// TwinCAT 3 PLC project TcAocLib
// Title: CNM AoC Lib
// Company: ekvip automation GmbH
// Author: tdie
// ProjectVersion: 0.0.0.0
// ProgramVersion: 3.1.4026.11
// libraries:
//   CNM_AbstractObject, * (ekvip automation GmbH)
//   CNM_AssertionInterfaceLib, * (ekvip automation GmbH)
//   CNM_CollectionInterfaces, * (ekvip automation GmbH)
//   CNM_Collections, * (ekvip automation GmbH)
//   CNM_CycleManager, * (ekvip automation GmbH)
//   CNM_CylceManagerInterfaces, * (ekvip automation GmbH)
//   CNM_ReturnTypes, * (ekvip automation GmbH)
//   CNM_UnicodeUtilities, * (ekvip automation GmbH)
//   Tc2_Standard, * (Beckhoff Automation GmbH)
//   Tc2_System, * (Beckhoff Automation GmbH)
//   Tc2_Utilities, * (Beckhoff Automation GmbH)
// project tree:
//   File/ FileHandler.TcPOU
//   Project Information/ F_GetCompany.TcPOU, F_GetTitle.TcPOU, F_GetVersion.TcPOU
//   Solver/ AbstractSolver.TcPOU
//   Strings/ GetAllLinesFromString.TcPOU, ILine.TcIO, IStringContainer.TcIO, Line.TcPOU
//   Strings/Wrapper/ ILineList.TcIO, IStringContainerList.TcIO, LineList.TcPOU, StringContainerList.TcPOU
//   Value/ IHaveUlintValue.TcIO, IHaveValue.TcIO, IHaveLintValue.TcIO, UlintValue.TcPOU, Value.TcPOU, ValueSum.TcPOU, LintValue.TcPOU
//   Version/ Global_Version.TcGVL
// (motion and I/O tree: see PLC project solutions)
// real-time tasks:
//   TASK PlcTask: cycle T#10ms, priority 20, ADS port 350

// ---- Version/Global_Version.TcGVL
{attribute 'TcGenerated'}
{attribute 'no-analysis'}
{attribute 'linkalways'}
// This function has been automatically generated from the project information.
VAR_GLOBAL CONSTANT
	{attribute 'const_non_replaced'}
	stLibVersion_CNM_AoC_Lib : ST_LibVersion := (iMajor := 0, iMinor := 0, iBuild := 0, iRevision := 0, nFlags := 0, sVersion := '0.0.0.0');
END_VAR

// ---- Strings/ILine.TcIO
INTERFACE ILine EXTENDS IStringContainer

METHOD splitBy : IStringContainerList
VAR_INPUT
	splitter	: STRING(255);
	addEmptyEntries :BOOL := FALSE;
END_VAR
END_METHOD

END_INTERFACE

// ---- Strings/IStringContainer.TcIO
INTERFACE IStringContainer EXTENDS IHaveValue

PROPERTY text : STRING(255)
GET
END_GET
SET
END_SET
END_PROPERTY

END_INTERFACE

// ---- Strings/Wrapper/ILineList.TcIO
INTERFACE ILineList EXTENDS CNM_AbstractObject.IObject

(*

short summary
=================
This methode adds the given CNM_AbstractObject.IObject to the end of the list.
Example: 
Given a list that looks like this: (Head->) A B C (<- End),
calling append(D) on this list will place the D at the and,
making it the new End: (Head->) A B C D(<- End)

.. <legal notes>

legal notes
=================
| SPDX-FileCopyrightText: © 2022 ekvip automation GmbH <info@ekvip.de>
| SPDX-License-Identifier: Apache-2.0
| For details check: Apache-2.0_

.. _Apache-2.0: https://www.apache.org/licenses/LICENSE-2.0

.. </legal notes>

parameters
=================

*)
METHOD append : CNM_CollectionInterfaces.CNM_ReturnTypes.SingleExecutionResult
VAR_INPUT
	(*The object to be appended*)
	line	: ILine;
END_VAR
END_METHOD

{warning 'Add method implementation '}
(*

short summary
=================
This methode adds all elements of the given collection to the end of this list.
Example:
For the list1: A B C and list2: D E F will be after list1.appendCollection(list2):
A B C D E F. Notice the elements are still in the same order they where befor on each subsection.

.. <legal notes>

legal notes
=================
| SPDX-FileCopyrightText: © 2022 ekvip automation GmbH <info@ekvip.de>
| SPDX-License-Identifier: Apache-2.0
| For details check: Apache-2.0_

.. _Apache-2.0: https://www.apache.org/licenses/LICENSE-2.0

.. </legal notes>

parameters
=================

*)
METHOD appendCollection : CNM_CollectionInterfaces.CNM_ReturnTypes.SingleExecutionResult
VAR_INPUT
	(*The collection to be appended*)
	collectionToAppend	: CNM_CollectionInterfaces.ICollection;
END_VAR
END_METHOD

{warning 'Add method implementation '}
(*

short summary
=================
This methode clears/deletes all clearable data from this object.
Example:
A list: 1 2 3 after list.clear() will have no remaining items, isEmpty = true.

.. <legal notes>

legal notes
=================
| SPDX-FileCopyrightText: © 2022 ekvip automation GmbH <info@ekvip.de>
| SPDX-License-Identifier: Apache-2.0
| For details check: Apache-2.0_

.. _Apache-2.0: https://www.apache.org/licenses/LICENSE-2.0

.. </legal notes>

parameters
=================

*)
METHOD clear
END_METHOD

{warning 'Add method implementation '}
(*

short summary
=================
This methode checks if a given object is contained in the collection. 
The object is inside if the collection contains an object where the default comperator of the objects returns EQUAL on compareTo!

.. <legal notes>

legal notes
=================
| SPDX-FileCopyrightText: © 2022 ekvip automation GmbH <info@ekvip.de>
| SPDX-License-Identifier: Apache-2.0
| For details check: Apache-2.0_

.. _Apache-2.0: https://www.apache.org/licenses/LICENSE-2.0

.. </legal notes>

parameters
=================
:return: ``FALSE``: list does not contain an equal object
    ``TRUE``: list does contain an equal object

*)
METHOD containsEqualLine : BOOL
VAR_INPUT
	(*the object to be checked if it exists inside the collection*)
	line	: ILine;
END_VAR
END_METHOD

{warning 'Add method implementation '}
(*

short summary
=================
This methode checks if a given object is contained in the collection. 
The object is inside if the collection contains an object of equal hashcode!

.. <legal notes>

legal notes
=================
| SPDX-FileCopyrightText: © 2022 ekvip automation GmbH <info@ekvip.de>
| SPDX-License-Identifier: Apache-2.0
| For details check: Apache-2.0_

.. _Apache-2.0: https://www.apache.org/licenses/LICENSE-2.0

.. </legal notes>

parameters
=================
:return: ``FALSE``: list does not contain given object,
    ``TRUE``: list does contain given object

*)
METHOD containsLine : BOOL
VAR_INPUT
	(*the object to be checked if it exists inside the collection*)
	line	: ILine;
END_VAR
END_METHOD

{warning 'Add method implementation '}
(*

short summary
=================
This property returns the last object in the first and removes it from the list. Can be seen as opposite of prepend.
Example:
On a list: (Head -->) A B C, list.dequeue will return A.
Example 2:
If you call prepend(x), a dequeue right after will return x.

.. <legal notes>

legal notes
=================
| SPDX-FileCopyrightText: © 2022 ekvip automation GmbH <info@ekvip.de>
| SPDX-License-Identifier: Apache-2.0
| For details check: Apache-2.0_

.. _Apache-2.0: https://www.apache.org/licenses/LICENSE-2.0

.. </legal notes>

*)
METHOD dequeue : ILine
END_METHOD

{warning 'Add method implementation '}
(*

short summary
=================
Method to perform a given action on all objects inside the collection.
Needs to reset the execution flag between calls.
Action to perform needs to implement :ref:`IApplier`.
Example:
You have a list of numbers: 1 2 3 and a ConcreteIncrementApplier that can take  a number and increment it. 
Calling list.forEach(TRUE, ConcreteIncrementApplier) will increment all numbers in the list, becoming: 2 3 4.

.. <legal notes>

legal notes
=================
| SPDX-FileCopyrightText: © 2022 ekvip automation GmbH <info@ekvip.de>
| SPDX-License-Identifier: Apache-2.0
| For details check: Apache-2.0_

.. _Apache-2.0: https://www.apache.org/licenses/LICENSE-2.0

.. </legal notes>

parameters
=========================
:return: CNM_ReturnTypes.ExecutionState

*)
METHOD forEach : CNM_CollectionInterfaces.CNM_ReturnTypes.SingleExecutionState
VAR_INPUT
	(*control bit to start or abort the forEach loop*)
	execute	: BOOL;
	(*the applier (action) to be used on all obejcts in the collection*)
	applier	: CNM_CollectionInterfaces.IApplier;
END_VAR
END_METHOD

{warning 'Add method implementation '}
(*

short summary
=================
This methode returns ths index of the first object that is equal to the given.
Example:
A list of: 1 2 3 after list.getIndexOf(1) will return: index=>0 and return IndexBounds.IN_BOUNDS
Example 2:
A list of: 1 2 3 after list.getIndexOf(4) will return: index=>3 and return IndexBounds.OUT_OF_BOUNDS

.. <legal notes>

legal notes
=================
| SPDX-FileCopyrightText: © 2022 ekvip automation GmbH <info@ekvip.de>
| SPDX-License-Identifier: Apache-2.0
| For details check: Apache-2.0_

.. _Apache-2.0: https://www.apache.org/licenses/LICENSE-2.0

.. </legal notes>

parameters
=================
:return: ``SingleExecutionResult.SUCCESS``: object found
    ``SingleExecutionResult.ERROR``: object couldn't be found in the list, index is undefined

*)
METHOD getIndexOf : CNM_CollectionInterfaces.CNM_ReturnTypes.SingleExecutionResult
VAR_INPUT
	(*the object to get the index from*)
	line	: ILine;
END_VAR
VAR_OUTPUT
	(*the index of the object inside the collection*)
	index	: __XWORD;
END_VAR
END_METHOD

{warning 'Add method implementation '}
(*

short summary
=================
This methode returns the object at the given index.
Returned objects can be modified, but not replaced! To replace an object use replaceObjectAt.
Example:
A list of: 1 2 3 after list.getObjectAt(1) will return: object=>2 and return SingleExecutionResult.SUCCESS
Example 2:
A list of: 1 2 3 after list.getObjectAt(3) will return: object=>NULL and return SingleExecutionResult.ERROR

.. <legal notes>

legal notes
=================
| SPDX-FileCopyrightText: © 2022 ekvip automation GmbH <info@ekvip.de>
| SPDX-License-Identifier: Apache-2.0
| For details check: Apache-2.0_

.. _Apache-2.0: https://www.apache.org/licenses/LICENSE-2.0

.. </legal notes>

parameters
=================
:return: ``SingleExecutionResult.SUCCESS``: index was valid
    ``SingleExecutionResult.ERROR``: index was not valid, returned object is undefined

*)
METHOD getLineAt : CNM_CollectionInterfaces.CNM_ReturnTypes.SingleExecutionResult
VAR_INPUT
	(*the index to access the object from*)
	index	: __XWORD;
END_VAR
VAR_OUTPUT
	(*the object at the given index*)
	line	: ILine;
END_VAR
END_METHOD

{warning 'Add property implementation'}
(*

short summary
=================
This property returns ``TRUE`` if the collection has any element.

.. <legal notes>

legal notes
=================
| SPDX-FileCopyrightText: © 2022 ekvip automation GmbH <info@ekvip.de>
| SPDX-License-Identifier: Apache-2.0
| For details check: Apache-2.0_

.. _Apache-2.0: https://www.apache.org/licenses/LICENSE-2.0

.. </legal notes>

*)
PROPERTY hasElement : BOOL
GET
END_GET
END_PROPERTY

{warning 'Add method implementation '}
(*

short summary
=================
This methode adds the given object at the given index. 
Will shift the other data starting at given index to the right.
List Lenght will be incremented.
Example:
A list of: 1 2 3 after list.insertObjectAt(1, object:=4) will become: 1 4 2 3 and return SingleExecutionResult.SUCCESS
Example 2:
A list of: 1 2 3 after list.insertObjectAt(3, object:=4) will become: 1 2 3 4 and return SingleExecutionResult.SUCCESS
Example 3:
A list of: 1 2 3 after list.insertObjectAt(5, object:=4) will become: 1 2 3 and return SingleExecutionResult.ERROR

.. <legal notes>

legal notes
=================
| SPDX-FileCopyrightText: © 2022 ekvip automation GmbH <info@ekvip.de>
| SPDX-License-Identifier: Apache-2.0
| For details check: Apache-2.0_

.. _Apache-2.0: https://www.apache.org/licenses/LICENSE-2.0

.. </legal notes>

parameters
=================
:return: ``SingleExecutionResult.SUCCESS``: index was valid, object inserted
    ``SingleExecutionResult.ERROR``: index out of bounds, list not changed

*)
METHOD insertLineAt : CNM_CollectionInterfaces.CNM_ReturnTypes.SingleExecutionResult
VAR_INPUT
	(*the index to insert the object at*)
	index	: __XWORD;
	(*the object to be added*)
	line	: ILine;
END_VAR
END_METHOD

{warning 'Add method implementation '}
(*

short summary
=================
This method sorts the Sortable in the inverted order, so from great to low
.. <legal notes>

legal notes
=================
| SPDX-FileCopyrightText: © 2022 ekvip automation GmbH <info@ekvip.de>
| SPDX-License-Identifier: Apache-2.0
| For details check: Apache-2.0_

.. _Apache-2.0: https://www.apache.org/licenses/LICENSE-2.0

.. </legal notes>

parameters
=========================
:return: ``ABORTED``: While inverse was pending,execute had a falling edge,
	``BUSY``: Inverse is in progress
	``ERROR``: Inverse was not able to finish (p.e. List changed) call inverse(false) to reset
	``IDLE``: Currently invert is not in progress
	``SUCCESS``: Inversing was finished 
*)
METHOD inverseSort : CNM_CollectionInterfaces.CNM_ReturnTypes.SingleExecutionState
VAR_INPUT
	(*control bit to start or abort the inverting, needs to be active until the ExecutionState is noz longer busy*)
	execute	: BOOL;
END_VAR
END_METHOD

{warning 'Add method implementation '}
(*

short summary
=================
Inverts the order of the elements inside the object. Does not apply any kind of sorting, only reverses.

.. <legal notes>

legal notes
=================
| SPDX-FileCopyrightText: © 2022 ekvip automation GmbH <info@ekvip.de>
| SPDX-License-Identifier: Apache-2.0
| For details check: Apache-2.0_

.. _Apache-2.0: https://www.apache.org/licenses/LICENSE-2.0

.. </legal notes>

parameters
=========================

*)
METHOD invert
END_METHOD

{warning 'Add property implementation'}
(*

short summary
=================
This property returns ``TRUE`` if the collection is empty.

.. <legal notes>

legal notes
=================
| SPDX-FileCopyrightText: © 2022 ekvip automation GmbH <info@ekvip.de>
| SPDX-License-Identifier: Apache-2.0
| For details check: Apache-2.0_

.. _Apache-2.0: https://www.apache.org/licenses/LICENSE-2.0

.. </legal notes>

*)
PROPERTY isEmpty : BOOL
GET
END_GET
END_PROPERTY

{warning 'Add method implementation '}
(*

short summary
=================
This methode returns the next object in the iteration and returns an execution state.
Example:
You have a list: 1 2 3
the first iterate call will return CNM_ReturnTypes.BUSY and object = 1
the second iterate call will return CNM_ReturnTypes.BUSY and object = 2
the third iterate call will return CNM_ReturnTypes.SUCCESS and object = 3

.. <legal notes>

legal notes
=================
| SPDX-FileCopyrightText: © 2022 ekvip automation GmbH <info@ekvip.de>
| SPDX-License-Identifier: Apache-2.0
| For details check: Apache-2.0_

.. _Apache-2.0: https://www.apache.org/licenses/LICENSE-2.0

.. </legal notes>

parameters
=================

*)
METHOD iterate : CNM_CollectionInterfaces.CNM_ReturnTypes.SingleExecutionState
VAR_INPUT
	(*control bit to start or abort the iterate*)
	execute	: BOOL;
END_VAR
VAR_OUTPUT
	(*the returned object of the iteration*)
	line	: ILine;
END_VAR
END_METHOD

{warning 'Add method implementation '}
(*

short summary
=================
This property returns the last object in the list and removes it from the list. Can be seen as opposite of append.
Example:
On a list: (Head -->) A B C, list.pop will return C.
Example 2:
If you call append(x), a pop right after will return x.
May return a null pointer if list is empty

.. <legal notes>

legal notes
=================
| SPDX-FileCopyrightText: © 2022 ekvip automation GmbH <info@ekvip.de>
| SPDX-License-Identifier: Apache-2.0
| For details check: Apache-2.0_

.. _Apache-2.0: https://www.apache.org/licenses/LICENSE-2.0

.. </legal notes>

*)
METHOD pop : ILine
END_METHOD

{warning 'Add method implementation '}
(*

short summary
=================
This methode adds the given obejct to the end of the list.
Example: 
Given a list that looks like this: (Head->) A B C (<- End),
calling prepend(D) on this list will place the D at start,
making it the new Head: (Head->) D A B C (<- End)

.. <legal notes>

legal notes
=================
| SPDX-FileCopyrightText: © 2022 ekvip automation GmbH <info@ekvip.de>
| SPDX-License-Identifier: Apache-2.0
| For details check: Apache-2.0_

.. _Apache-2.0: https://www.apache.org/licenses/LICENSE-2.0

.. </legal notes>

parameters
=================
:return: ``SingleExecutionResult.SUCCESS``: prepend was successful
	``SingleExecutionResult.ERROR``: allocation of memory for new object failed
	
*)
METHOD prepend : CNM_CollectionInterfaces.CNM_ReturnTypes.SingleExecutionResult
VAR_INPUT
	(*The object to be prepended*)
	line	: ILine;
END_VAR
END_METHOD

{warning 'Add method implementation '}
(*

short summary
=================
This methode adds all elements of the given collection to the start of this list. 
Example:
For the list1: A B C and list2: D E F will be after list1.prependCollection(list2):
D E F A B C. Notice the elements are still in the same order they where befor on each subsection.

.. <legal notes>

legal notes
=================
| SPDX-FileCopyrightText: © 2022 ekvip automation GmbH <info@ekvip.de>
| SPDX-License-Identifier: Apache-2.0
| For details check: Apache-2.0_

.. _Apache-2.0: https://www.apache.org/licenses/LICENSE-2.0

.. </legal notes>

parameters
=================
:return: ``SingleExecutionResult.SUCCESS``: prependCollection was successful
	``SingleExecutionResult.ERROR``: could not allocate memory for all new elements, list is left unchanged

*)
METHOD prependCollection : CNM_CollectionInterfaces.CNM_ReturnTypes.SingleExecutionResult
VAR_INPUT
	(*The collection to be prepended*)
	collectionToPrepend	: CNM_CollectionInterfaces.ICollection;
END_VAR
END_METHOD

{warning 'Add method implementation '}
(*

short summary
=================
This methode removes the first instance of the given object from the list.
Compares objects with hash value.
For example a Linked List: A B C A A D will on remove(A) becomes: B C A A D

.. <legal notes>

legal notes
=================
| SPDX-FileCopyrightText: © 2022 ekvip automation GmbH <info@ekvip.de>
| SPDX-License-Identifier: Apache-2.0
| For details check: Apache-2.0_

.. _Apache-2.0: https://www.apache.org/licenses/LICENSE-2.0

.. </legal notes>

parameters
=================

*)
METHOD remove
VAR_INPUT
	(*The object to be removed from the list*)
	line	: ILine;
END_VAR
END_METHOD

{warning 'Add method implementation '}
(*

short summary
=================
This methode removes the element at the given index. 
Will shift the remaining data to the left (no empty space in list)
List Length will be decremented.
Example:
A list of: 1 2 3 after list.removeObjectAt(1) will become: 1 3 and return IndexBounds.IN_BOUNDS
Example 2:
A list of: 1 2 3 after list.removeObjectAt(3) will reamin: 1 2 3 and return IndexBounds.OUT_OF_BOUNDS

.. <legal notes>

legal notes
=================
| SPDX-FileCopyrightText: © 2022 ekvip automation GmbH <info@ekvip.de>
| SPDX-License-Identifier: Apache-2.0
| For details check: Apache-2.0_

.. _Apache-2.0: https://www.apache.org/licenses/LICENSE-2.0

.. </legal notes>

parameters
=================
:return: ``SingleExecutionResult.SUCCESS``: Element removed from index
    ``SingleExecutionResult.ERROR``: index out of bound, no object removed

*)
METHOD removeLineAt : CNM_CollectionInterfaces.CNM_ReturnTypes.SingleExecutionResult
VAR_INPUT
	(*the index to remove the object from*)
	index	: __XWORD;
END_VAR
END_METHOD

{warning 'Add method implementation '}
(*

short summary
=================
This methode replaces the Interface reference inside the collection at the given index with the given Interface.
Example:
A list of: 1 2 3 after list.replaceObjectAt(1, withObject:=4) will become: 1 4 3 and return SingleExecutionResult.SUCCESS
Example 2:
A list of: 1 2 3 after list.replaceObjectAt(3, withObject:=4) will remain: 1 2 3 and return SingleExecutionResult.ERROR

.. <legal notes>

legal notes
=================
| SPDX-FileCopyrightText: © 2022 ekvip automation GmbH <info@ekvip.de>
| SPDX-License-Identifier: Apache-2.0
| For details check: Apache-2.0_

.. _Apache-2.0: https://www.apache.org/licenses/LICENSE-2.0

.. </legal notes>

parameters
=================
:return: ``SingleExecutionResult.SUCCESS``: index valid, element at index replaced with ``withObject``
    ``SingleExecutionResult.ERROR``: ìndex out of bounds, nothing changed

*)
METHOD replaceLineAt : CNM_CollectionInterfaces.CNM_ReturnTypes.SingleExecutionResult
VAR_INPUT
	(*the index to replace the object at*)
	index	: __XWORD;
	(*the object to be at this index instead*)
	withLine	: ILine;
END_VAR
END_METHOD

{warning 'Add method implementation '}
(*

short summary
=================
This methode can replace the default sorter for a custom one. Check :ref:`IListSorter`
Can be used for performant sorting algorithms if more about the data structure is known.

.. attention:: 
	For implementations: **IListSorter is an empty interface and you should extend it with custom interfaces for each type of list.**
	For LinkedList see :ref:`ILinkedListSorter`. 
	Your implementation should then use this extended interface and the setter should check for compability. 
	
.. <legal notes>

legal notes
=================
| SPDX-FileCopyrightText: © 2022 ekvip automation GmbH <info@ekvip.de>
| SPDX-License-Identifier: Apache-2.0
| For details check: Apache-2.0_

.. _Apache-2.0: https://www.apache.org/licenses/LICENSE-2.0

.. </legal notes>

parameters
=================
:return: ``THIS^`` :ref:`IList`

*)
METHOD setSorter : CNM_CollectionInterfaces.ISortable
VAR_INPUT
	(*The instance of the sorter to be used to sort the list*)
	sorter	: CNM_CollectionInterfaces.IArrayListSorter;
END_VAR
END_METHOD

{warning 'Add property implementation'}
(*

short summary
=================
This property returns the number of elements inside this collection.

.. <legal notes>

legal notes
=================
| SPDX-FileCopyrightText: © 2022 ekvip automation GmbH <info@ekvip.de>
| SPDX-License-Identifier: Apache-2.0
| For details check: Apache-2.0_

.. _Apache-2.0: https://www.apache.org/licenses/LICENSE-2.0

.. </legal notes>

*)
PROPERTY size : __XWORD
GET
END_GET
END_PROPERTY

{warning 'Add method implementation '}
(*

short summary
=================
This method sorts the data structure. 
This can take many cycles and should be called until the CNM_ReturnTypes.ExecutionState is no longer ``BUSY``.

.. <legal notes>

legal notes
=================
| SPDX-FileCopyrightText: © 2022 ekvip automation GmbH <info@ekvip.de>
| SPDX-License-Identifier: Apache-2.0
| For details check: Apache-2.0_

.. _Apache-2.0: https://www.apache.org/licenses/LICENSE-2.0

.. </legal notes>

parameters
=================
:return: ``ABORTED``: While sort was pending,execute had a falling edge,
	``BUSY``: Sort is in progress
	``ERROR``: Sort was not able to finish (p.e. List changed) call sort(false) to reset
	``IDLE``: Currently no sort in progress
	``SUCCESS``: Sorting was finished 

*)
METHOD sort : CNM_CollectionInterfaces.CNM_ReturnTypes.SingleExecutionState
VAR_INPUT
	(*control bit to start or abort the sorting, needs to be active until the ExecutionState is SUCCESS*)
	execute	: BOOL;
END_VAR
END_METHOD

{warning 'Add method implementation '}
(*

short summary
=================
This method sorts the data structure. 
It uses the passed Comperator to sort the structure.
This can take many cycles and should be called until the CNM_ReturnTypes.ExecutionState is no longer ``BUSY``.

.. <legal notes>

legal notes
=================
| SPDX-FileCopyrightText: © 2022 ekvip automation GmbH <info@ekvip.de>
| SPDX-License-Identifier: Apache-2.0
| For details check: Apache-2.0_

.. _Apache-2.0: https://www.apache.org/licenses/LICENSE-2.0

.. </legal notes>

parameters
=================
:return: ``ABORTED``: While sort was pending,execute had a falling edge,
	``BUSY``: Sort is in progress
	``ERROR``: Sort was not able to finish (p.e. List changed) call sort(false) to reset
	``IDLE``: Currently no sort in progress
	``SUCCESS``: Sorting was finished 

*)
METHOD sortWithComparator : CNM_CollectionInterfaces.CNM_ReturnTypes.SingleExecutionState
VAR_INPUT
	(*control bit to start or abort the sorting, needs to be active until the ExecutionState is SUCCESS*)
	execute	: BOOL;
	(*the comparator that should be used for the sort. Must not be changed while sort is in process*)
	comparator	: CNM_CollectionInterfaces.CNM_AbstractObject.IComparator;
END_VAR
END_METHOD

END_INTERFACE

// ---- Strings/Wrapper/IStringContainerList.TcIO
INTERFACE IStringContainerList EXTENDS CNM_AbstractObject.IObject

(*

short summary
=================
This methode adds the given CNM_AbstractObject.IObject to the end of the list.
Example: 
Given a list that looks like this: (Head->) A B C (<- End),
calling append(D) on this list will place the D at the and,
making it the new End: (Head->) A B C D(<- End)

.. <legal notes>

legal notes
=================
| SPDX-FileCopyrightText: © 2022 ekvip automation GmbH <info@ekvip.de>
| SPDX-License-Identifier: Apache-2.0
| For details check: Apache-2.0_

.. _Apache-2.0: https://www.apache.org/licenses/LICENSE-2.0

.. </legal notes>

parameters
=================

*)
METHOD append : CNM_CollectionInterfaces.CNM_ReturnTypes.SingleExecutionResult
VAR_INPUT
	(*The object to be appended*)
	stringcontainer	: IStringContainer;
END_VAR
END_METHOD

{warning 'Add method implementation '}
(*

short summary
=================
This methode adds all elements of the given collection to the end of this list.
Example:
For the list1: A B C and list2: D E F will be after list1.appendCollection(list2):
A B C D E F. Notice the elements are still in the same order they where befor on each subsection.

.. <legal notes>

legal notes
=================
| SPDX-FileCopyrightText: © 2022 ekvip automation GmbH <info@ekvip.de>
| SPDX-License-Identifier: Apache-2.0
| For details check: Apache-2.0_

.. _Apache-2.0: https://www.apache.org/licenses/LICENSE-2.0

.. </legal notes>

parameters
=================

*)
METHOD appendCollection : CNM_CollectionInterfaces.CNM_ReturnTypes.SingleExecutionResult
VAR_INPUT
	(*The collection to be appended*)
	collectionToAppend	: CNM_CollectionInterfaces.ICollection;
END_VAR
END_METHOD

{warning 'Add method implementation '}
(*

short summary
=================
This methode clears/deletes all clearable data from this object.
Example:
A list: 1 2 3 after list.clear() will have no remaining items, isEmpty = true.

.. <legal notes>

legal notes
=================
| SPDX-FileCopyrightText: © 2022 ekvip automation GmbH <info@ekvip.de>
| SPDX-License-Identifier: Apache-2.0
| For details check: Apache-2.0_

.. _Apache-2.0: https://www.apache.org/licenses/LICENSE-2.0

.. </legal notes>

parameters
=================

*)
METHOD clear
END_METHOD

{warning 'Add method implementation '}
(*

short summary
=================
This methode checks if a given object is contained in the collection. 
The object is inside if the collection contains an object where the default comperator of the objects returns EQUAL on compareTo!

.. <legal notes>

legal notes
=================
| SPDX-FileCopyrightText: © 2022 ekvip automation GmbH <info@ekvip.de>
| SPDX-License-Identifier: Apache-2.0
| For details check: Apache-2.0_

.. _Apache-2.0: https://www.apache.org/licenses/LICENSE-2.0

.. </legal notes>

parameters
=================
:return: ``FALSE``: list does not contain an equal object
    ``TRUE``: list does contain an equal object

*)
METHOD containsEqualStringContainer : BOOL
VAR_INPUT
	(*the object to be checked if it exists inside the collection*)
	stringcontainer	: IStringContainer;
END_VAR
END_METHOD

{warning 'Add method implementation '}
(*

short summary
=================
This methode checks if a given object is contained in the collection. 
The object is inside if the collection contains an object of equal hashcode!

.. <legal notes>

legal notes
=================
| SPDX-FileCopyrightText: © 2022 ekvip automation GmbH <info@ekvip.de>
| SPDX-License-Identifier: Apache-2.0
| For details check: Apache-2.0_

.. _Apache-2.0: https://www.apache.org/licenses/LICENSE-2.0

.. </legal notes>

parameters
=================
:return: ``FALSE``: list does not contain given object,
    ``TRUE``: list does contain given object

*)
METHOD containsStringContainer : BOOL
VAR_INPUT
	(*the object to be checked if it exists inside the collection*)
	stringcontainer	: IStringContainer;
END_VAR
END_METHOD

{warning 'Add method implementation '}
(*

short summary
=================
This property returns the last object in the first and removes it from the list. Can be seen as opposite of prepend.
Example:
On a list: (Head -->) A B C, list.dequeue will return A.
Example 2:
If you call prepend(x), a dequeue right after will return x.

.. <legal notes>

legal notes
=================
| SPDX-FileCopyrightText: © 2022 ekvip automation GmbH <info@ekvip.de>
| SPDX-License-Identifier: Apache-2.0
| For details check: Apache-2.0_

.. _Apache-2.0: https://www.apache.org/licenses/LICENSE-2.0

.. </legal notes>

*)
METHOD dequeue : IStringContainer
END_METHOD

{warning 'Add method implementation '}
(*

short summary
=================
Method to perform a given action on all objects inside the collection.
Needs to reset the execution flag between calls.
Action to perform needs to implement :ref:`IApplier`.
Example:
You have a list of numbers: 1 2 3 and a ConcreteIncrementApplier that can take  a number and increment it. 
Calling list.forEach(TRUE, ConcreteIncrementApplier) will increment all numbers in the list, becoming: 2 3 4.

.. <legal notes>

legal notes
=================
| SPDX-FileCopyrightText: © 2022 ekvip automation GmbH <info@ekvip.de>
| SPDX-License-Identifier: Apache-2.0
| For details check: Apache-2.0_

.. _Apache-2.0: https://www.apache.org/licenses/LICENSE-2.0

.. </legal notes>

parameters
=========================
:return: CNM_ReturnTypes.ExecutionState

*)
METHOD forEach : CNM_CollectionInterfaces.CNM_ReturnTypes.SingleExecutionState
VAR_INPUT
	(*control bit to start or abort the forEach loop*)
	execute	: BOOL;
	(*the applier (action) to be used on all obejcts in the collection*)
	applier	: CNM_CollectionInterfaces.IApplier;
END_VAR
END_METHOD

{warning 'Add method implementation '}
(*

short summary
=================
This methode returns ths index of the first object that is equal to the given.
Example:
A list of: 1 2 3 after list.getIndexOf(1) will return: index=>0 and return IndexBounds.IN_BOUNDS
Example 2:
A list of: 1 2 3 after list.getIndexOf(4) will return: index=>3 and return IndexBounds.OUT_OF_BOUNDS

.. <legal notes>

legal notes
=================
| SPDX-FileCopyrightText: © 2022 ekvip automation GmbH <info@ekvip.de>
| SPDX-License-Identifier: Apache-2.0
| For details check: Apache-2.0_

.. _Apache-2.0: https://www.apache.org/licenses/LICENSE-2.0

.. </legal notes>

parameters
=================
:return: ``SingleExecutionResult.SUCCESS``: object found
    ``SingleExecutionResult.ERROR``: object couldn't be found in the list, index is undefined

*)
METHOD getIndexOf : CNM_CollectionInterfaces.CNM_ReturnTypes.SingleExecutionResult
VAR_INPUT
	(*the object to get the index from*)
	stringcontainer	: IStringContainer;
END_VAR
VAR_OUTPUT
	(*the index of the object inside the collection*)
	index	: __XWORD;
END_VAR
END_METHOD

{warning 'Add method implementation '}
(*

short summary
=================
This methode returns the object at the given index.
Returned objects can be modified, but not replaced! To replace an object use replaceObjectAt.
Example:
A list of: 1 2 3 after list.getObjectAt(1) will return: object=>2 and return SingleExecutionResult.SUCCESS
Example 2:
A list of: 1 2 3 after list.getObjectAt(3) will return: object=>NULL and return SingleExecutionResult.ERROR

.. <legal notes>

legal notes
=================
| SPDX-FileCopyrightText: © 2022 ekvip automation GmbH <info@ekvip.de>
| SPDX-License-Identifier: Apache-2.0
| For details check: Apache-2.0_

.. _Apache-2.0: https://www.apache.org/licenses/LICENSE-2.0

.. </legal notes>

parameters
=================
:return: ``SingleExecutionResult.SUCCESS``: index was valid
    ``SingleExecutionResult.ERROR``: index was not valid, returned object is undefined

*)
METHOD getStringContainerAt : CNM_CollectionInterfaces.CNM_ReturnTypes.SingleExecutionResult
VAR_INPUT
	(*the index to access the object from*)
	index	: __XWORD;
END_VAR
VAR_OUTPUT
	(*the object at the given index*)
	stringcontainer	: IStringContainer;
END_VAR
END_METHOD

{warning 'Add property implementation'}
(*

short summary
=================
This property returns ``TRUE`` if the collection has any element.

.. <legal notes>

legal notes
=================
| SPDX-FileCopyrightText: © 2022 ekvip automation GmbH <info@ekvip.de>
| SPDX-License-Identifier: Apache-2.0
| For details check: Apache-2.0_

.. _Apache-2.0: https://www.apache.org/licenses/LICENSE-2.0

.. </legal notes>

*)
PROPERTY hasElement : BOOL
GET
END_GET
END_PROPERTY

{warning 'Add method implementation '}
(*

short summary
=================
This methode adds the given object at the given index. 
Will shift the other data starting at given index to the right.
List Lenght will be incremented.
Example:
A list of: 1 2 3 after list.insertObjectAt(1, object:=4) will become: 1 4 2 3 and return SingleExecutionResult.SUCCESS
Example 2:
A list of: 1 2 3 after list.insertObjectAt(3, object:=4) will become: 1 2 3 4 and return SingleExecutionResult.SUCCESS
Example 3:
A list of: 1 2 3 after list.insertObjectAt(5, object:=4) will become: 1 2 3 and return SingleExecutionResult.ERROR

.. <legal notes>

legal notes
=================
| SPDX-FileCopyrightText: © 2022 ekvip automation GmbH <info@ekvip.de>
| SPDX-License-Identifier: Apache-2.0
| For details check: Apache-2.0_

.. _Apache-2.0: https://www.apache.org/licenses/LICENSE-2.0

.. </legal notes>

parameters
=================
:return: ``SingleExecutionResult.SUCCESS``: index was valid, object inserted
    ``SingleExecutionResult.ERROR``: index out of bounds, list not changed

*)
METHOD insertStringContainerAt : CNM_CollectionInterfaces.CNM_ReturnTypes.SingleExecutionResult
VAR_INPUT
	(*the index to insert the object at*)
	index	: __XWORD;
	(*the object to be added*)
	stringcontainer	: IStringContainer;
END_VAR
END_METHOD

{warning 'Add method implementation '}
(*

short summary
=================
This method sorts the Sortable in the inverted order, so from great to low
.. <legal notes>

legal notes
=================
| SPDX-FileCopyrightText: © 2022 ekvip automation GmbH <info@ekvip.de>
| SPDX-License-Identifier: Apache-2.0
| For details check: Apache-2.0_

.. _Apache-2.0: https://www.apache.org/licenses/LICENSE-2.0

.. </legal notes>

parameters
=========================
:return: ``ABORTED``: While inverse was pending,execute had a falling edge,
	``BUSY``: Inverse is in progress
	``ERROR``: Inverse was not able to finish (p.e. List changed) call inverse(false) to reset
	``IDLE``: Currently invert is not in progress
	``SUCCESS``: Inversing was finished 
*)
METHOD inverseSort : CNM_CollectionInterfaces.CNM_ReturnTypes.SingleExecutionState
VAR_INPUT
	(*control bit to start or abort the inverting, needs to be active until the ExecutionState is noz longer busy*)
	execute	: BOOL;
END_VAR
END_METHOD

{warning 'Add method implementation '}
(*

short summary
=================
Inverts the order of the elements inside the object. Does not apply any kind of sorting, only reverses.

.. <legal notes>

legal notes
=================
| SPDX-FileCopyrightText: © 2022 ekvip automation GmbH <info@ekvip.de>
| SPDX-License-Identifier: Apache-2.0
| For details check: Apache-2.0_

.. _Apache-2.0: https://www.apache.org/licenses/LICENSE-2.0

.. </legal notes>

parameters
=========================

*)
METHOD invert
END_METHOD

{warning 'Add property implementation'}
(*

short summary
=================
This property returns ``TRUE`` if the collection is empty.

.. <legal notes>

legal notes
=================
| SPDX-FileCopyrightText: © 2022 ekvip automation GmbH <info@ekvip.de>
| SPDX-License-Identifier: Apache-2.0
| For details check: Apache-2.0_

.. _Apache-2.0: https://www.apache.org/licenses/LICENSE-2.0

.. </legal notes>

*)
PROPERTY isEmpty : BOOL
GET
END_GET
END_PROPERTY

{warning 'Add method implementation '}
(*

short summary
=================
This methode returns the next object in the iteration and returns an execution state.
Example:
You have a list: 1 2 3
the first iterate call will return CNM_ReturnTypes.BUSY and object = 1
the second iterate call will return CNM_ReturnTypes.BUSY and object = 2
the third iterate call will return CNM_ReturnTypes.SUCCESS and object = 3

.. <legal notes>

legal notes
=================
| SPDX-FileCopyrightText: © 2022 ekvip automation GmbH <info@ekvip.de>
| SPDX-License-Identifier: Apache-2.0
| For details check: Apache-2.0_

.. _Apache-2.0: https://www.apache.org/licenses/LICENSE-2.0

.. </legal notes>

parameters
=================

*)
METHOD iterate : CNM_CollectionInterfaces.CNM_ReturnTypes.SingleExecutionState
VAR_INPUT
	(*control bit to start or abort the iterate*)
	execute	: BOOL;
END_VAR
VAR_OUTPUT
	(*the returned object of the iteration*)
	stringcontainer	: IStringContainer;
END_VAR
END_METHOD

{warning 'Add method implementation '}
(*

short summary
=================
This property returns the last object in the list and removes it from the list. Can be seen as opposite of append.
Example:
On a list: (Head -->) A B C, list.pop will return C.
Example 2:
If you call append(x), a pop right after will return x.
May return a null pointer if list is empty

.. <legal notes>

legal notes
=================
| SPDX-FileCopyrightText: © 2022 ekvip automation GmbH <info@ekvip.de>
| SPDX-License-Identifier: Apache-2.0
| For details check: Apache-2.0_

.. _Apache-2.0: https://www.apache.org/licenses/LICENSE-2.0

.. </legal notes>

*)
METHOD pop : IStringContainer
END_METHOD

{warning 'Add method implementation '}
(*

short summary
=================
This methode adds the given obejct to the end of the list.
Example: 
Given a list that looks like this: (Head->) A B C (<- End),
calling prepend(D) on this list will place the D at start,
making it the new Head: (Head->) D A B C (<- End)

.. <legal notes>

legal notes
=================
| SPDX-FileCopyrightText: © 2022 ekvip automation GmbH <info@ekvip.de>
| SPDX-License-Identifier: Apache-2.0
| For details check: Apache-2.0_

.. _Apache-2.0: https://www.apache.org/licenses/LICENSE-2.0

.. </legal notes>

parameters
=================
:return: ``SingleExecutionResult.SUCCESS``: prepend was successful
	``SingleExecutionResult.ERROR``: allocation of memory for new object failed
	
*)
METHOD prepend : CNM_CollectionInterfaces.CNM_ReturnTypes.SingleExecutionResult
VAR_INPUT
	(*The object to be prepended*)
	stringcontainer	: IStringContainer;
END_VAR
END_METHOD

{warning 'Add method implementation '}
(*

short summary
=================
This methode adds all elements of the given collection to the start of this list. 
Example:
For the list1: A B C and list2: D E F will be after list1.prependCollection(list2):
D E F A B C. Notice the elements are still in the same order they where befor on each subsection.

.. <legal notes>

legal notes
=================
| SPDX-FileCopyrightText: © 2022 ekvip automation GmbH <info@ekvip.de>
| SPDX-License-Identifier: Apache-2.0
| For details check: Apache-2.0_

.. _Apache-2.0: https://www.apache.org/licenses/LICENSE-2.0

.. </legal notes>

parameters
=================
:return: ``SingleExecutionResult.SUCCESS``: prependCollection was successful
	``SingleExecutionResult.ERROR``: could not allocate memory for all new elements, list is left unchanged

*)
METHOD prependCollection : CNM_CollectionInterfaces.CNM_ReturnTypes.SingleExecutionResult
VAR_INPUT
	(*The collection to be prepended*)
	collectionToPrepend	: CNM_CollectionInterfaces.ICollection;
END_VAR
END_METHOD

{warning 'Add method implementation '}
(*

short summary
=================
This methode removes the first instance of the given object from the list.
Compares objects with hash value.
For example a Linked List: A B C A A D will on remove(A) becomes: B C A A D

.. <legal notes>

legal notes
=================
| SPDX-FileCopyrightText: © 2022 ekvip automation GmbH <info@ekvip.de>
| SPDX-License-Identifier: Apache-2.0
| For details check: Apache-2.0_

.. _Apache-2.0: https://www.apache.org/licenses/LICENSE-2.0

.. </legal notes>

parameters
=================

*)
METHOD remove
VAR_INPUT
	(*The object to be removed from the list*)
	stringcontainer	: IStringContainer;
END_VAR
END_METHOD

{warning 'Add method implementation '}
(*

short summary
=================
This methode removes the element at the given index. 
Will shift the remaining data to the left (no empty space in list)
List Length will be decremented.
Example:
A list of: 1 2 3 after list.removeObjectAt(1) will become: 1 3 and return IndexBounds.IN_BOUNDS
Example 2:
A list of: 1 2 3 after list.removeObjectAt(3) will reamin: 1 2 3 and return IndexBounds.OUT_OF_BOUNDS

.. <legal notes>

legal notes
=================
| SPDX-FileCopyrightText: © 2022 ekvip automation GmbH <info@ekvip.de>
| SPDX-License-Identifier: Apache-2.0
| For details check: Apache-2.0_

.. _Apache-2.0: https://www.apache.org/licenses/LICENSE-2.0

.. </legal notes>

parameters
=================
:return: ``SingleExecutionResult.SUCCESS``: Element removed from index
    ``SingleExecutionResult.ERROR``: index out of bound, no object removed

*)
METHOD removeStringContainerAt : CNM_CollectionInterfaces.CNM_ReturnTypes.SingleExecutionResult
VAR_INPUT
	(*the index to remove the object from*)
	index	: __XWORD;
END_VAR
END_METHOD

{warning 'Add method implementation '}
(*

short summary
=================
This methode replaces the Interface reference inside the collection at the given index with the given Interface.
Example:
A list of: 1 2 3 after list.replaceObjectAt(1, withObject:=4) will become: 1 4 3 and return SingleExecutionResult.SUCCESS
Example 2:
A list of: 1 2 3 after list.replaceObjectAt(3, withObject:=4) will remain: 1 2 3 and return SingleExecutionResult.ERROR

.. <legal notes>

legal notes
=================
| SPDX-FileCopyrightText: © 2022 ekvip automation GmbH <info@ekvip.de>
| SPDX-License-Identifier: Apache-2.0
| For details check: Apache-2.0_

.. _Apache-2.0: https://www.apache.org/licenses/LICENSE-2.0

.. </legal notes>

parameters
=================
:return: ``SingleExecutionResult.SUCCESS``: index valid, element at index replaced with ``withObject``
    ``SingleExecutionResult.ERROR``: ìndex out of bounds, nothing changed

*)
METHOD replaceStringContainerAt : CNM_CollectionInterfaces.CNM_ReturnTypes.SingleExecutionResult
VAR_INPUT
	(*the index to replace the object at*)
	index	: __XWORD;
	(*the object to be at this index instead*)
	withStringContainer	: IStringContainer;
END_VAR
END_METHOD

{warning 'Add method implementation '}
(*

short summary
=================
This methode can replace the default sorter for a custom one. Check :ref:`IListSorter`
Can be used for performant sorting algorithms if more about the data structure is known.

.. attention:: 
	For implementations: **IListSorter is an empty interface and you should extend it with custom interfaces for each type of list.**
	For LinkedList see :ref:`ILinkedListSorter`. 
	Your implementation should then use this extended interface and the setter should check for compability. 
	
.. <legal notes>

legal notes
=================
| SPDX-FileCopyrightText: © 2022 ekvip automation GmbH <info@ekvip.de>
| SPDX-License-Identifier: Apache-2.0
| For details check: Apache-2.0_

.. _Apache-2.0: https://www.apache.org/licenses/LICENSE-2.0

.. </legal notes>

parameters
=================
:return: ``THIS^`` :ref:`IList`

*)
METHOD setSorter : CNM_CollectionInterfaces.ISortable
VAR_INPUT
	(*The instance of the sorter to be used to sort the list*)
	sorter	: CNM_CollectionInterfaces.IArrayListSorter;
END_VAR
END_METHOD

{warning 'Add property implementation'}
(*

short summary
=================
This property returns the number of elements inside this collection.

.. <legal notes>

legal notes
=================
| SPDX-FileCopyrightText: © 2022 ekvip automation GmbH <info@ekvip.de>
| SPDX-License-Identifier: Apache-2.0
| For details check: Apache-2.0_

.. _Apache-2.0: https://www.apache.org/licenses/LICENSE-2.0

.. </legal notes>

*)
PROPERTY size : __XWORD
GET
END_GET
END_PROPERTY

{warning 'Add method implementation '}
(*

short summary
=================
This method sorts the data structure. 
This can take many cycles and should be called until the CNM_ReturnTypes.ExecutionState is no longer ``BUSY``.

.. <legal notes>

legal notes
=================
| SPDX-FileCopyrightText: © 2022 ekvip automation GmbH <info@ekvip.de>
| SPDX-License-Identifier: Apache-2.0
| For details check: Apache-2.0_

.. _Apache-2.0: https://www.apache.org/licenses/LICENSE-2.0

.. </legal notes>

parameters
=================
:return: ``ABORTED``: While sort was pending,execute had a falling edge,
	``BUSY``: Sort is in progress
	``ERROR``: Sort was not able to finish (p.e. List changed) call sort(false) to reset
	``IDLE``: Currently no sort in progress
	``SUCCESS``: Sorting was finished 

*)
METHOD sort : CNM_CollectionInterfaces.CNM_ReturnTypes.SingleExecutionState
VAR_INPUT
	(*control bit to start or abort the sorting, needs to be active until the ExecutionState is SUCCESS*)
	execute	: BOOL;
END_VAR
END_METHOD

{warning 'Add method implementation '}
(*

short summary
=================
This method sorts the data structure. 
It uses the passed Comperator to sort the structure.
This can take many cycles and should be called until the CNM_ReturnTypes.ExecutionState is no longer ``BUSY``.

.. <legal notes>

legal notes
=================
| SPDX-FileCopyrightText: © 2022 ekvip automation GmbH <info@ekvip.de>
| SPDX-License-Identifier: Apache-2.0
| For details check: Apache-2.0_

.. _Apache-2.0: https://www.apache.org/licenses/LICENSE-2.0

.. </legal notes>

parameters
=================
:return: ``ABORTED``: While sort was pending,execute had a falling edge,
	``BUSY``: Sort is in progress
	``ERROR``: Sort was not able to finish (p.e. List changed) call sort(false) to reset
	``IDLE``: Currently no sort in progress
	``SUCCESS``: Sorting was finished 

*)
METHOD sortWithComparator : CNM_CollectionInterfaces.CNM_ReturnTypes.SingleExecutionState
VAR_INPUT
	(*control bit to start or abort the sorting, needs to be active until the ExecutionState is SUCCESS*)
	execute	: BOOL;
	(*the comparator that should be used for the sort. Must not be changed while sort is in process*)
	comparator	: CNM_CollectionInterfaces.CNM_AbstractObject.IComparator;
END_VAR
END_METHOD

END_INTERFACE

// ---- Value/IHaveUlintValue.TcIO
(*
	dont we all?
*)
INTERFACE IHaveUlintValue EXTENDS CNM_AbstractObject.IObject

PROPERTY value : ULINT
GET
END_GET
SET
END_SET
END_PROPERTY

END_INTERFACE

// ---- Value/IHaveValue.TcIO
(*
	dont we all?
*)
INTERFACE IHaveValue EXTENDS CNM_AbstractObject.IObject

PROPERTY value : LREAL
GET
END_GET
SET
END_SET
END_PROPERTY

END_INTERFACE

// ---- Value/IHaveLintValue.TcIO
(*
	dont we all?
*)
INTERFACE IHaveLintValue EXTENDS CNM_AbstractObject.IObject

PROPERTY value : LINT
GET
END_GET
SET
END_SET
END_PROPERTY

END_INTERFACE

// ---- File/FileHandler.TcPOU
FUNCTION_BLOCK FileHandler
VAR_INPUT
END_VAR
VAR_OUTPUT
END_VAR
VAR
	fbFileOpen		:FB_FileOpen;	
	fbFileClose		:FB_FileClose;	
	writer		:FB_FileWrite;
	reader :FB_FileRead;
END_VAR

Global.TC_EVENTS.AocError.ParseError;

METHOD read : SingleExecutionState
VAR_INPUT
	execute			: BOOL;	(* Rising edge starts program execution *)
	text :POINTER TO BYTE;
	sNetId			: T_AmsNetId;		(* TwinCAT system network address *)
	sDirectoryPath	: T_MaxString;		(* CSV destination directory path e.g. 'C:/temp/' *)
	sFileName		: T_MaxString;		(* CSV destination file name e.g. 'Dividos' automatically extended by a timestamp *)
	readLen : UDINT;
END_VAR
VAR_INST
	cm :CNM_CycleManager.SimpleCycleManager();
	hFile			: UINT		:= 0;	(* File handle of the source file *)
END_VAR
VAR
	busy			: BOOL;
	bError			: BOOL;
	nErrId			: UDINT;
	writeString 		: STRING(255);
END_VAR
VAR CONSTANT
	STATE_OPEN_SOURCE_FILE	: INT := 2;
	STATE_WAIT_FILE_OPENED	: INT := 3;
	STATE_READ				: INT := 4;
	STATE_READ_FINISHED	: INT := 5;
	STATE_CLOSE_SOURCE_FILE	: INT := 6;
	STATE_WAIT_FILE_CLOSED	: INT := 7;
	STATE_ERROR				: INT := 100;
END_VAR
cm(execute := execute);

CASE cm.step.current OF
CNM_ReturnTypes.DefaultSteps.STEP.IDLE:;
CNM_ReturnTypes.DefaultSteps.STEP.INIT:
	busy 	:= TRUE;
	bError	:= FALSE;
	nErrId	:= 0;
	cm.proceed();

STATE_OPEN_SOURCE_FILE:	(* Open source file *)
	fbFileOpen( 
		sNetId := sNetId, 
		sPathName := Tc2_Standard.CONCAT(Tc2_Standard.CONCAT(sDirectoryPath, '\'), sFileName),
		nMode := Tc2_System.Global_Variables.FOPEN_MODEREAD OR Tc2_System.Global_Variables.FOPEN_MODETEXT,(* Open file in TEXT mode! *)
		ePath := PATH_GENERIC, 
		hFile => hFile,
		bExecute := cm.executeStep,
		bBusy => busy
	);
	cm.waitFor(NOT busy);

STATE_WAIT_FILE_OPENED:
	IF NOT fbFileOpen.bError THEN
		cm.proceed();
	ELSE(* Error: file not found? *)
		cm.evaluate(state := CNM_ReturnTypes.SingleExecutionState.ERROR);
	END_IF

STATE_READ:
	reader(
		sNetId := sNetId, 
		hFile := hFile, 
		pReadBuff := text,
		bExecute := cm.executeStep,
		cbReadLen := readLen,
		bBusy => busy,
	);
	cm.waitFor(NOT busy);

STATE_READ_FINISHED:	(* Wait until write not busy *)
	IF NOT writer.bError THEN
		cm.proceed();
	ELSE(* Error: file not found? *)
		cm.proceedWith(STATE_CLOSE_SOURCE_FILE);
	END_IF

STATE_CLOSE_SOURCE_FILE:	(* Close source file *)
	fbFileClose( 
		sNetId := sNetId, 
		hFile := hFile, 
		bExecute := cm.executeStep,
		bBusy => busy
	);
	cm.waitFor(NOT busy);

STATE_WAIT_FILE_CLOSED:(* Wait until close not busy *)
	IF NOT fbFileClose.bError THEN
		cm.proceedWith(CNM_ReturnTypes.DefaultSteps.STEP.SUCCESS);
	ELSE(* Error: file not found? *)
		cm.evaluate(state := CNM_ReturnTypes.SingleExecutionState.ERROR);
	END_IF
	
CNM_ReturnTypes.DefaultSteps.STEP.ERROR:;
CNM_ReturnTypes.DefaultSteps.STEP.SUCCESS:;
END_CASE

read := cm.state;
END_METHOD

METHOD write : CNM_ReturnTypes.SingleExecutionState
VAR_INPUT
	execute			: BOOL;	(* Rising edge starts program execution *)
	text :POINTER TO BYTE;
	sNetId			: T_AmsNetId;		(* TwinCAT system network address *)
	sDirectoryPath	: T_MaxString;		(* CSV destination directory path e.g. 'C:/temp/' *)
	sFileName		: T_MaxString;		(* CSV destination file name e.g. 'Dividos' automatically extended by a timestamp *)
END_VAR
VAR_INST
	cm :CNM_CycleManager.SimpleCycleManager();
	hFile			: UINT		:= 0;	(* File handle of the source file *)
END_VAR
VAR
	busy			: BOOL;
	bError			: BOOL;
	nErrId			: UDINT;
	writeString 		: STRING(255);
END_VAR
VAR CONSTANT
	STATE_OPEN_SOURCE_FILE	: INT := 2;
	STATE_WAIT_FILE_OPENED	: INT := 3;
	STATE_WRITE				: INT := 4;
	STATE_WRITE_FINISHED	: INT := 5;
	STATE_CLOSE_SOURCE_FILE	: INT := 6;
	STATE_WAIT_FILE_CLOSED	: INT := 7;
	STATE_ERROR				: INT := 100;
END_VAR
cm(execute := execute);

CASE cm.step.current OF
CNM_ReturnTypes.DefaultSteps.STEP.IDLE:;
CNM_ReturnTypes.DefaultSteps.STEP.INIT:
	busy 	:= FALSE;
	bError	:= FALSE;
	nErrId	:= 0;
	cm.proceed();

STATE_OPEN_SOURCE_FILE:	(* Open source file *)
	fbFileOpen( 
		sNetId := sNetId, 
		sPathName := Tc2_Standard.CONCAT(Tc2_Standard.CONCAT(sDirectoryPath, '\'), sFileName),
		nMode := FOPEN_MODEAPPEND OR FOPEN_MODETEXT,(* Open file in TEXT mode! *)
		ePath := PATH_GENERIC, 
		hFile => hFile,
		bExecute := cm.executeStep,
		bBusy => busy
	);
	cm.waitFor(NOT busy);

STATE_WAIT_FILE_OPENED:
	IF NOT fbFileOpen.bError THEN
		cm.proceed();
	ELSE(* Error: file not found? *)
		cm.evaluate(state := CNM_ReturnTypes.SingleExecutionState.ERROR);
	END_IF

STATE_WRITE:
	writer(
		sNetId := sNetId, 
		hFile := hFile, 
		pWriteBuff := text, 
		cbWriteLen := LEN2(text), 
		bExecute := cm.executeStep,
		bBusy => busy
	);
	cm.waitFor(NOT busy);

STATE_WRITE_FINISHED:	(* Wait until write not busy *)
	IF NOT writer.bError THEN
		cm.proceed();
	ELSE(* Error: file not found? *)
		cm.proceedWith(STATE_CLOSE_SOURCE_FILE);
	END_IF

STATE_CLOSE_SOURCE_FILE:	(* Close source file *)
	fbFileClose( 
		sNetId := sNetId, 
		hFile := hFile, 
		bExecute := cm.executeStep,
		bBusy => busy
	);
	cm.waitFor(NOT busy);

STATE_WAIT_FILE_CLOSED:(* Wait until close not busy *)
	IF NOT fbFileClose.bError THEN
		cm.proceedWith(CNM_ReturnTypes.DefaultSteps.STEP.SUCCESS);
	ELSE(* Error: file not found? *)
		cm.evaluate(state := CNM_ReturnTypes.SingleExecutionState.ERROR);
	END_IF
	
CNM_ReturnTypes.DefaultSteps.STEP.ERROR:;
CNM_ReturnTypes.DefaultSteps.STEP.SUCCESS:;
END_CASE

write := cm.state;
END_METHOD

END_FUNCTION_BLOCK

// ---- Project Information/F_GetCompany.TcPOU
// This function has been automatically generated from the project information.
{attribute 'signature_flag' := '1073741824'}
{attribute 'TcGenerated'}
{attribute 'no-analysis'}
FUNCTION F_GetCompany : WSTRING
VAR_INPUT
	
END_VAR

F_GetCompany := "ekvip automation GmbH";

END_FUNCTION

// ---- Project Information/F_GetTitle.TcPOU
// This function has been automatically generated from the project information.
{attribute 'signature_flag' := '1073741824'}
{attribute 'TcGenerated'}
{attribute 'no-analysis'}
FUNCTION F_GetTitle : WSTRING
VAR_INPUT
	
END_VAR

F_GetTitle := "CNM AoC Lib";

END_FUNCTION

// ---- Project Information/F_GetVersion.TcPOU
// This function has been automatically generated from the project information.
{attribute 'signature_flag' := '1073741824'}
{attribute 'TcGenerated'}
{attribute 'no-analysis'}
FUNCTION F_GetVersion : ST_LibVersion
VAR_INPUT
	
END_VAR

F_GetVersion.iMajor := 0;
F_GetVersion.iMinor := 0;
F_GetVersion.iBuild := 0;
F_GetVersion.iRevision := 0;
F_GetVersion.sVersion := '0.0.0.0';
F_GetVersion.nFlags := 0;

END_FUNCTION

// ---- Solver/AbstractSolver.TcPOU
FUNCTION_BLOCK ABSTRACT AbstractSolver
VAR
	io :FileHandler();
	bufferRead : STRING(64000) := '';
	bufferWrite : STRING(255) := '';	
	cm :CNM_CycleManager.SimpleCycleManager();
	lines :ILineList;
	inoutPath : STRING;
	snetId :STRING;	
	inputFile :STRING;
	outputFile :STRING := 'solution.txt';
END_VAR

//FB_Init is always available implicitly and it is used primarily for initialization.
//The return value is not evaluated. For a specific influence, you can also declare the
//methods explicitly and provide additional code there with the standard initialization
//code. You can evaluate the return value.
METHOD FB_Init: BOOL
VAR_INPUT
    bInitRetains: BOOL; // TRUE: the retain variables are initialized (reset warm / reset cold)
    bInCopyCode: BOOL;  // TRUE: the instance will be copied to the copy code afterward (online change)
	sNetId :STRING;   
	folderPath :STRING;   
	inputFile :STRING;   
	outputFile :STRING;   
END_VAR
THIS^.snetId := sNetId;
THIS^.inoutPath := folderPath;
THIS^.inputFile := inputFile;
THIS^.outputFile := outputFile;
END_METHOD

METHOD FINAL run : CNM_ReturnTypes.SingleExecutionState
VAR_INPUT
	execute :BOOL;
END_VAR
VAR CONSTANT
	READ_INPUT :DINT := 2;
	GET_LINES :DINT := READ_INPUT + 1;
END_VAR
cm(execute := execute);

CASE cm.step.current OF
CNM_ReturnTypes.DefaultSteps.STEP.IDLE:;
CNM_ReturnTypes.DefaultSteps.STEP.INIT:
	cm.waitFor(inoutPath <> '' AND snetId <> '');
READ_INPUT:
	cm.evaluate(
		io.read(
			execute := cm.executeStep, 
			text := ADR(bufferRead), 
			sNetId := THIS^.snetId, 
			sDirectoryPath := THIS^.inoutPath, 
			sFileName := THIS^.inputFile,
			readLen := SIZEOF(THIS^.bufferRead)
		)
	);
GET_LINES:
	lines := GetAllLinesFromString(ADR(THIS^.bufferRead), SIZEOF(THIS^.bufferRead));
	cm.proceed();
CNM_ReturnTypes.DefaultSteps.STEP.SUCCESS:;
CNM_ReturnTypes.DefaultSteps.STEP.ERROR:;
ELSE
	THIS^.solve(cm.step.current);
END_CASE
END_METHOD

METHOD ABSTRACT solve
VAR_INPUT
	step :DINT;
END_VAR
END_METHOD

METHOD FINAL writeSolution
cm.evaluate(
	io.write(
		execute := cm.executeStep, 
		text := ADR(THIS^.bufferWrite), 
		sNetId := THIS^.snetId, 
		sDirectoryPath := THIS^.inoutPath, 
		sFileName := THIS^.outputFile
	)
);
END_METHOD

END_FUNCTION_BLOCK

// ---- Strings/GetAllLinesFromString.TcPOU
FUNCTION GetAllLinesFromString :ILineList
VAR_INPUT
	text :POINTER TO BYTE;
	textSize :UDINT;
	addEmptyLines : BOOL := FALSE;
END_VAR
VAR
	index : UDINT;
	startLineIndex : UDINT;
	currentLineText : STRING(255);
	currentLine :ILine;
	currentLineObject :IObject;
	pCurrentLine :POINTER TO Line;
	pList :POINTER TO LineList;
END_VAR

pList := __NEW(LineList());

FOR index := 0 TO textSize DO
	startLineIndex := index;
	IF(text[index] = 0)THEN
		EXIT;
	END_IF
	WHILE(index < textSize)DO
		IF(text[index] = 10 OR text[index] = 0)THEN //10 is newLine $N
			IF(index - startLineIndex > 255)THEN
				EXIT;
			END_IF 
			Tc2_System.MEMSET(ADR(currentLineText), 0, SIZEOF(currentLineText));
			Tc2_System.MEMCPY(ADR(currentLineText), text+startLineIndex, index - startLineIndex);
			IF(Tc2_Standard.LEN(currentLineText) = 0 AND NOT addEmptyLines)THEN
				EXIT;
			END_IF
			pCurrentLine := __NEW(Line());
			pCurrentLine^.text := currentLineText;
			pList^.append(pCurrentLine^);
			EXIT;
		END_IF
		index := index+1;
	END_WHILE
END_FOR

GetAllLinesFromString := pList^;

END_FUNCTION

// ---- Strings/Line.TcPOU
{attribute 'enable_dynamic_creation'}
FUNCTION_BLOCK Line EXTENDS Object IMPLEMENTS ILine
VAR_INPUT
END_VAR
VAR_OUTPUT
END_VAR
VAR
	content :STRING(255);
	number :LREAL;
END_VAR

(*

short summary
=================
This abstract property returns the class name of the concrete object, 
which is useful for logging/debugging purpose or to check the class name
for ``__DELETE`` in factories (sometimes it's necessary to do more 
than just to free the memory).

.. <legal notes>

legal notes
=================
| SPDX-FileCopyrightText: © 2022 ekvip automation GmbH <info@ekvip.de>
| SPDX-License-Identifier: Apache-2.0
| For details check: Apache-2.0_

.. _Apache-2.0: https://www.apache.org/licenses/LICENSE-2.0

.. </legal notes>

*)
PROPERTY className : CNM_AbstractObject.ClassName
GET
END_GET
END_PROPERTY

METHOD splitBy :IStringContainerList
VAR_INPUT
	splitter	: STRING(255);
	addEmptyEntries :BOOL := FALSE;
END_VAR
VAR
	pContainterList :POINTER TO StringContainerList;
	
	index :INT;
	searchindex :INT;
	textSize :INT;
	splitterSize :INT;
	lastSplit :INT;
	startSearchIndex : UDINT;
	pContainer :POINTER TO Line;
	currentText : STRING(255);
END_VAR
splitterSize := Tc2_Standard.LEN(splitter);
textSize := Tc2_Standard.LEN(THIS^.text);

pContainterList := __NEW(StringContainerList());
splitBy := pContainterList^;

RETURN (splitterSize = 0);

lastSplit := 0;
FOR index := 0 TO textSize DO
	startSearchIndex := index;
	searchindex := 0;
	WHILE(startSearchIndex+searchindex < textSize AND_THEN THIS^.content[startSearchIndex+searchindex] = splitter[searchindex])DO
		IF(searchindex = splitterSize)THEN //10 is newLine $N
			Tc2_System.MEMSET(ADR(currentText), 0, SIZEOF(currentText));
			Tc2_System.MEMCPY(ADR(currentText), ADR(THIS^.content)+startSearchIndex+searchindex, startSearchIndex + searchindex - splitterSize);
			IF(Tc2_Standard.LEN(currentText) = 0 AND NOT addEmptyEntries)THEN
				index := index + searchindex;
				EXIT;
			END_IF
			pContainer := __NEW(Line());
			pContainer^.text := currentText;
			splitBy.append(pContainer^);
			index := index + searchindex;
			lastSplit := index;
			EXIT;
		END_IF
		searchindex := searchindex+1;
	END_WHILE
END_FOR

Tc2_System.MEMSET(ADR(currentText), 0, SIZEOF(currentText));
Tc2_System.MEMCPY(ADR(currentText), ADR(THIS^.content) + lastSplit, index - lastSplit);
IF(Tc2_Standard.LEN(currentText) = 0 AND NOT addEmptyEntries)THEN
	RETURN;
END_IF
pContainer := __NEW(Line());
pContainer^.text := currentText;
splitBy.append(pContainer^);
END_METHOD

PROPERTY text : STRING(255)
GET
text := THIS^.content;
END_GET
SET
THIS^.content := text;
END_SET
END_PROPERTY

PROPERTY value : LREAL
GET
value := THIS^.number;
END_GET
SET
THIS^.number := value;
END_SET
END_PROPERTY

END_FUNCTION_BLOCK

// ---- Strings/Wrapper/StringContainerList.TcPOU
{attribute 'enable_dynamic_creation'}
FUNCTION_BLOCK StringContainerList EXTENDS CNM_AbstractObject.Object IMPLEMENTS IStringContainerList
VAR
	list : CNM_Collections.ArrayList(1000);
END_VAR

(*

short summary
=================
This methode adds the given CNM_AbstractObject.IObject to the end of the list.
Example: 
Given a list that looks like this: (Head->) A B C (<- End),
calling append(D) on this list will place the D at the and,
making it the new End: (Head->) A B C D(<- End)

.. <legal notes>

legal notes
=================
| SPDX-FileCopyrightText: © 2022 ekvip automation GmbH <info@ekvip.de>
| SPDX-License-Identifier: Apache-2.0
| For details check: Apache-2.0_

.. _Apache-2.0: https://www.apache.org/licenses/LICENSE-2.0

.. </legal notes>

parameters
=================

*)
METHOD append : CNM_ReturnTypes.SingleExecutionResult
VAR_INPUT
	(*The object to be appended*)
	stringcontainer	: IStringContainer;
END_VAR
append := THIS^.list.append(object := stringcontainer);
END_METHOD

(*

short summary
=================
This methode adds all elements of the given collection to the end of this list.
Example:
For the list1: A B C and list2: D E F will be after list1.appendCollection(list2):
A B C D E F. Notice the elements are still in the same order they where befor on each subsection.

.. <legal notes>

legal notes
=================
| SPDX-FileCopyrightText: © 2022 ekvip automation GmbH <info@ekvip.de>
| SPDX-License-Identifier: Apache-2.0
| For details check: Apache-2.0_

.. _Apache-2.0: https://www.apache.org/licenses/LICENSE-2.0

.. </legal notes>

parameters
=================

*)
METHOD appendCollection : CNM_ReturnTypes.SingleExecutionResult
VAR_INPUT
	(*The collection to be appended*)
	collectionToAppend	: CNM_CollectionInterfaces.ICollection;
END_VAR
appendCollection := THIS^.list.appendCollection(collectionToAppend);
END_METHOD

PROPERTY className : ClassName
GET
className := 'StringContainerList';
END_GET
END_PROPERTY

(*

short summary
=================
This methode clears/deletes all clearable data from this object.
Example:
A list: 1 2 3 after list.clear() will have no remaining items, isEmpty = true.

.. <legal notes>

legal notes
=================
| SPDX-FileCopyrightText: © 2022 ekvip automation GmbH <info@ekvip.de>
| SPDX-License-Identifier: Apache-2.0
| For details check: Apache-2.0_

.. _Apache-2.0: https://www.apache.org/licenses/LICENSE-2.0

.. </legal notes>

parameters
=================

*)
METHOD clear
THIS^.list.clear();
END_METHOD

(*

short summary
=================
This methode checks if a given object is contained in the collection. 
The object is inside if the collection contains an object where the default comperator of the objects returns EQUAL on compareTo!

.. <legal notes>

legal notes
=================
| SPDX-FileCopyrightText: © 2022 ekvip automation GmbH <info@ekvip.de>
| SPDX-License-Identifier: Apache-2.0
| For details check: Apache-2.0_

.. _Apache-2.0: https://www.apache.org/licenses/LICENSE-2.0

.. </legal notes>

parameters
=================
:return: ``FALSE``: list does not contain an equal object
    ``TRUE``: list does contain an equal object

*)
METHOD containsEqualStringContainer : BOOL
VAR_INPUT
	(*the object to be checked if it exists inside the collection*)
	stringcontainer	: IStringContainer;
END_VAR
containsEqualStringContainer := THIS^.list.containsEqualObject(object := stringcontainer);
END_METHOD

(*

short summary
=================
This methode checks if a given object is contained in the collection. 
The object is inside if the collection contains an object of equal hashcode!

.. <legal notes>

legal notes
=================
| SPDX-FileCopyrightText: © 2022 ekvip automation GmbH <info@ekvip.de>
| SPDX-License-Identifier: Apache-2.0
| For details check: Apache-2.0_

.. _Apache-2.0: https://www.apache.org/licenses/LICENSE-2.0

.. </legal notes>

parameters
=================
:return: ``FALSE``: list does not contain given object,
    ``TRUE``: list does contain given object

*)
METHOD containsStringContainer : BOOL
VAR_INPUT
	(*the object to be checked if it exists inside the collection*)
	stringcontainer	: IStringContainer;
END_VAR
containsStringContainer := THIS^.list.containsObject(object := stringcontainer);
END_METHOD

{warning 'Add method implementation '}
(*

short summary
=================
This method is a self-destruction if the object was created dynamically.
If the object is a container class, the container content is destroyed with it.
The output NULL is a constant which is always NULL,
this allows a semi-pleasant notation: ``foo.deepDestruct(NULL => foo);``.

.. <legal notes>

legal notes
=================
| SPDX-FileCopyrightText: © 2022 ekvip automation GmbH <info@ekvip.de>
| SPDX-License-Identifier: Apache-2.0
| For details check: Apache-2.0_

.. _Apache-2.0: https://www.apache.org/licenses/LICENSE-2.0

.. </legal notes>

parameters
=================

InOut:
	+-----------------+------+---------+------------------------------------------+
	| Scope           | Name | Type    | Comment                                  |
	+=================+======+=========+==========================================+
	| Output CONSTANT | NULL | __XWORD | ``NULL`` is a constant which is always 0 |
	+-----------------+------+---------+------------------------------------------+

*)
METHOD deepDestruct
VAR_OUTPUT CONSTANT
	(* NULL is a constant which is always 0 *)
	NULL	: __XWORD;
END_VAR
THIS^.list.deepDestruct();
END_METHOD

(*

short summary
=================
This property returns the last object in the first and removes it from the list. Can be seen as opposite of prepend.
Example:
On a list: (Head -->) A B C, list.dequeue will return A.
Example 2:
If you call prepend(x), a dequeue right after will return x.

.. <legal notes>

legal notes
=================
| SPDX-FileCopyrightText: © 2022 ekvip automation GmbH <info@ekvip.de>
| SPDX-License-Identifier: Apache-2.0
| For details check: Apache-2.0_

.. _Apache-2.0: https://www.apache.org/licenses/LICENSE-2.0

.. </legal notes>

*)
METHOD dequeue : IStringContainer
__QUERYINTERFACE(THIS^.list.dequeue(), dequeue);
END_METHOD

(*

short summary
=================
Method to perform a given action on all objects inside the collection.
Needs to reset the execution flag between calls.
Action to perform needs to implement :ref:`IApplier`.
Example:
You have a list of numbers: 1 2 3 and a ConcreteIncrementApplier that can take  a number and increment it. 
Calling list.forEach(TRUE, ConcreteIncrementApplier) will increment all numbers in the list, becoming: 2 3 4.

.. <legal notes>

legal notes
=================
| SPDX-FileCopyrightText: © 2022 ekvip automation GmbH <info@ekvip.de>
| SPDX-License-Identifier: Apache-2.0
| For details check: Apache-2.0_

.. _Apache-2.0: https://www.apache.org/licenses/LICENSE-2.0

.. </legal notes>

parameters
=========================
:return: CNM_ReturnTypes.ExecutionState

*)
METHOD forEach : CNM_ReturnTypes.SingleExecutionState
VAR_INPUT
	(*control bit to start or abort the forEach loop*)
	execute	: BOOL;
	(*the applier (action) to be used on all obejcts in the collection*)
	applier	: CNM_CollectionInterfaces.IApplier;
END_VAR
forEach := THIS^.list.forEach.parallel(execute := execute, applier := applier);
END_METHOD

(*

short summary
=================
This methode returns ths index of the first object that is equal to the given.
Example:
A list of: 1 2 3 after list.getIndexOf(1) will return: index=>0 and return IndexBounds.IN_BOUNDS
Example 2:
A list of: 1 2 3 after list.getIndexOf(4) will return: index=>3 and return IndexBounds.OUT_OF_BOUNDS

.. <legal notes>

legal notes
=================
| SPDX-FileCopyrightText: © 2022 ekvip automation GmbH <info@ekvip.de>
| SPDX-License-Identifier: Apache-2.0
| For details check: Apache-2.0_

.. _Apache-2.0: https://www.apache.org/licenses/LICENSE-2.0

.. </legal notes>

parameters
=================
:return: ``SingleExecutionResult.SUCCESS``: object found
    ``SingleExecutionResult.ERROR``: object couldn't be found in the list, index is undefined

*)
METHOD getIndexOf : CNM_ReturnTypes.SingleExecutionResult
VAR_INPUT
	(*the object to get the index from*)
	stringcontainer	: IStringContainer;
END_VAR
VAR_OUTPUT
	(*the index of the object inside the collection*)
	index	: __XWORD;
END_VAR
getIndexOf := THIS^.list.getIndexOf(object := stringcontainer, index => index);
END_METHOD

(*

short summary
=================
This methode returns the object at the given index.
Returned objects can be modified, but not replaced! To replace an object use replaceObjectAt.
Example:
A list of: 1 2 3 after list.getObjectAt(1) will return: object=>2 and return SingleExecutionResult.SUCCESS
Example 2:
A list of: 1 2 3 after list.getObjectAt(3) will return: object=>NULL and return SingleExecutionResult.ERROR

.. <legal notes>

legal notes
=================
| SPDX-FileCopyrightText: © 2022 ekvip automation GmbH <info@ekvip.de>
| SPDX-License-Identifier: Apache-2.0
| For details check: Apache-2.0_

.. _Apache-2.0: https://www.apache.org/licenses/LICENSE-2.0

.. </legal notes>

parameters
=================
:return: ``SingleExecutionResult.SUCCESS``: index was valid
    ``SingleExecutionResult.ERROR``: index was not valid, returned object is undefined

*)
METHOD getStringContainerAt : CNM_ReturnTypes.SingleExecutionResult
VAR_INPUT
	(*the index to access the object from*)
	index	: __XWORD;
END_VAR
VAR_OUTPUT
	(*the object at the given index*)
	stringcontainer	: IStringContainer;
END_VAR
VAR
	tmp : IObject;
END_VAR
getStringContainerAt := THIS^.list.getObjectAt(index := index, object => tmp);
__QUERYINTERFACE(tmp, stringcontainer);
END_METHOD

(*

short summary
=================
This property returns ``TRUE`` if the collection has any element.

.. <legal notes>

legal notes
=================
| SPDX-FileCopyrightText: © 2022 ekvip automation GmbH <info@ekvip.de>
| SPDX-License-Identifier: Apache-2.0
| For details check: Apache-2.0_

.. _Apache-2.0: https://www.apache.org/licenses/LICENSE-2.0

.. </legal notes>

*)
PROPERTY hasElement : BOOL
GET
hasElement := this^.list.hasElement;
END_GET
END_PROPERTY

(*

short summary
=================
This methode adds the given object at the given index. 
Will shift the other data starting at given index to the right.
List Lenght will be incremented.
Example:
A list of: 1 2 3 after list.insertObjectAt(1, object:=4) will become: 1 4 2 3 and return SingleExecutionResult.SUCCESS
Example 2:
A list of: 1 2 3 after list.insertObjectAt(3, object:=4) will become: 1 2 3 4 and return SingleExecutionResult.SUCCESS
Example 3:
A list of: 1 2 3 after list.insertObjectAt(5, object:=4) will become: 1 2 3 and return SingleExecutionResult.ERROR

.. <legal notes>

legal notes
=================
| SPDX-FileCopyrightText: © 2022 ekvip automation GmbH <info@ekvip.de>
| SPDX-License-Identifier: Apache-2.0
| For details check: Apache-2.0_

.. _Apache-2.0: https://www.apache.org/licenses/LICENSE-2.0

.. </legal notes>

parameters
=================
:return: ``SingleExecutionResult.SUCCESS``: index was valid, object inserted
    ``SingleExecutionResult.ERROR``: index out of bounds, list not changed

*)
METHOD insertStringContainerAt : CNM_ReturnTypes.SingleExecutionResult
VAR_INPUT
	(*the index to insert the object at*)
	index	: __XWORD;
	(*the object to be added*)
	stringcontainer	: IStringContainer;
END_VAR
insertStringContainerAt := THIS^.list.insertObjectAt(index := index, object := stringcontainer);
END_METHOD

(*

short summary
=================
This method sorts the Sortable in the inverted order, so from great to low
.. <legal notes>

legal notes
=================
| SPDX-FileCopyrightText: © 2022 ekvip automation GmbH <info@ekvip.de>
| SPDX-License-Identifier: Apache-2.0
| For details check: Apache-2.0_

.. _Apache-2.0: https://www.apache.org/licenses/LICENSE-2.0

.. </legal notes>

parameters
=========================
:return: ``ABORTED``: While inverse was pending,execute had a falling edge,
	``BUSY``: Inverse is in progress
	``ERROR``: Inverse was not able to finish (p.e. List changed) call inverse(false) to reset
	``IDLE``: Currently invert is not in progress
	``SUCCESS``: Inversing was finished 
*)
METHOD inverseSort : CNM_ReturnTypes.SingleExecutionState
VAR_INPUT
	(*control bit to start or abort the inverting, needs to be active until the ExecutionState is noz longer busy*)
	execute	: BOOL;
END_VAR
inverseSort := THIS^.list.inverseSort(execute := execute);
END_METHOD

(*

short summary
=================
Inverts the order of the elements inside the object. Does not apply any kind of sorting, only reverses.

.. <legal notes>

legal notes
=================
| SPDX-FileCopyrightText: © 2022 ekvip automation GmbH <info@ekvip.de>
| SPDX-License-Identifier: Apache-2.0
| For details check: Apache-2.0_

.. _Apache-2.0: https://www.apache.org/licenses/LICENSE-2.0

.. </legal notes>

parameters
=========================

*)
METHOD invert
THIS^.list.invert();
END_METHOD

(*

short summary
=================
This property returns ``TRUE`` if the collection is empty.

.. <legal notes>

legal notes
=================
| SPDX-FileCopyrightText: © 2022 ekvip automation GmbH <info@ekvip.de>
| SPDX-License-Identifier: Apache-2.0
| For details check: Apache-2.0_

.. _Apache-2.0: https://www.apache.org/licenses/LICENSE-2.0

.. </legal notes>

*)
PROPERTY isEmpty : BOOL
GET
isEmpty := THIS^.list.isEmpty;
END_GET
END_PROPERTY

(*

short summary
=================
This methode returns the next object in the iteration and returns an execution state.
Example:
You have a list: 1 2 3
the first iterate call will return CNM_ReturnTypes.BUSY and object = 1
the second iterate call will return CNM_ReturnTypes.BUSY and object = 2
the third iterate call will return CNM_ReturnTypes.SUCCESS and object = 3

.. <legal notes>

legal notes
=================
| SPDX-FileCopyrightText: © 2022 ekvip automation GmbH <info@ekvip.de>
| SPDX-License-Identifier: Apache-2.0
| For details check: Apache-2.0_

.. _Apache-2.0: https://www.apache.org/licenses/LICENSE-2.0

.. </legal notes>

parameters
=================

*)
METHOD iterate : CNM_ReturnTypes.SingleExecutionState
VAR_INPUT
	(*control bit to start or abort the iterate*)
	execute	: BOOL;
END_VAR
VAR_OUTPUT
	(*the returned object of the iteration*)
	stringcontainer	: IStringContainer;
END_VAR
VAR
	tmp : IObject;
END_VAR
iterate := THIS^.list.iterate(execute := execute, object => tmp);
__QUERYINTERFACE(tmp, stringcontainer);
END_METHOD

(*

short summary
=================
This property returns the last object in the list and removes it from the list. Can be seen as opposite of append.
Example:
On a list: (Head -->) A B C, list.pop will return C.
Example 2:
If you call append(x), a pop right after will return x.
May return a null pointer if list is empty

.. <legal notes>

legal notes
=================
| SPDX-FileCopyrightText: © 2022 ekvip automation GmbH <info@ekvip.de>
| SPDX-License-Identifier: Apache-2.0
| For details check: Apache-2.0_

.. _Apache-2.0: https://www.apache.org/licenses/LICENSE-2.0

.. </legal notes>

*)
METHOD pop : IStringContainer
__QUERYINTERFACE(THIS^.list.pop(), pop);
END_METHOD

(*

short summary
=================
This methode adds the given obejct to the end of the list.
Example: 
Given a list that looks like this: (Head->) A B C (<- End),
calling prepend(D) on this list will place the D at start,
making it the new Head: (Head->) D A B C (<- End)

.. <legal notes>

legal notes
=================
| SPDX-FileCopyrightText: © 2022 ekvip automation GmbH <info@ekvip.de>
| SPDX-License-Identifier: Apache-2.0
| For details check: Apache-2.0_

.. _Apache-2.0: https://www.apache.org/licenses/LICENSE-2.0

.. </legal notes>

parameters
=================
:return: ``SingleExecutionResult.SUCCESS``: prepend was successful
	``SingleExecutionResult.ERROR``: allocation of memory for new object failed
	
*)
METHOD prepend : CNM_ReturnTypes.SingleExecutionResult
VAR_INPUT
	(*The object to be prepended*)
	stringcontainer	: IStringContainer;
END_VAR
prepend := THIS^.list.prepend(object := stringcontainer);
END_METHOD

(*

short summary
=================
This methode adds all elements of the given collection to the start of this list. 
Example:
For the list1: A B C and list2: D E F will be after list1.prependCollection(list2):
D E F A B C. Notice the elements are still in the same order they where befor on each subsection.

.. <legal notes>

legal notes
=================
| SPDX-FileCopyrightText: © 2022 ekvip automation GmbH <info@ekvip.de>
| SPDX-License-Identifier: Apache-2.0
| For details check: Apache-2.0_

.. _Apache-2.0: https://www.apache.org/licenses/LICENSE-2.0

.. </legal notes>

parameters
=================
:return: ``SingleExecutionResult.SUCCESS``: prependCollection was successful
	``SingleExecutionResult.ERROR``: could not allocate memory for all new elements, list is left unchanged

*)
METHOD prependCollection : CNM_ReturnTypes.SingleExecutionResult
VAR_INPUT
	(*The collection to be prepended*)
	collectionToPrepend	: CNM_CollectionInterfaces.ICollection;
END_VAR
prependCollection := THIS^.list.prependCollection(collectionToPrepend := collectionToPrepend);
END_METHOD

(*

short summary
=================
This methode removes the first instance of the given object from the list.
Compares objects with hash value.
For example a Linked List: A B C A A D will on remove(A) becomes: B C A A D

.. <legal notes>

legal notes
=================
| SPDX-FileCopyrightText: © 2022 ekvip automation GmbH <info@ekvip.de>
| SPDX-License-Identifier: Apache-2.0
| For details check: Apache-2.0_

.. _Apache-2.0: https://www.apache.org/licenses/LICENSE-2.0

.. </legal notes>

parameters
=================

*)
METHOD remove
VAR_INPUT
	(*The object to be removed from the list*)
	stringcontainer	: IStringContainer;
END_VAR
THIS^.list.remove(object := stringcontainer);
END_METHOD

(*

short summary
=================
This methode removes the element at the given index. 
Will shift the remaining data to the left (no empty space in list)
List Length will be decremented.
Example:
A list of: 1 2 3 after list.removeObjectAt(1) will become: 1 3 and return IndexBounds.IN_BOUNDS
Example 2:
A list of: 1 2 3 after list.removeObjectAt(3) will reamin: 1 2 3 and return IndexBounds.OUT_OF_BOUNDS

.. <legal notes>

legal notes
=================
| SPDX-FileCopyrightText: © 2022 ekvip automation GmbH <info@ekvip.de>
| SPDX-License-Identifier: Apache-2.0
| For details check: Apache-2.0_

.. _Apache-2.0: https://www.apache.org/licenses/LICENSE-2.0

.. </legal notes>

parameters
=================
:return: ``SingleExecutionResult.SUCCESS``: Element removed from index
    ``SingleExecutionResult.ERROR``: index out of bound, no object removed

*)
METHOD removeStringContainerAt : CNM_ReturnTypes.SingleExecutionResult
VAR_INPUT
	(*the index to remove the object from*)
	index	: __XWORD;
END_VAR
removeStringContainerAt := THIS^.list.removeObjectAt(index := index);
END_METHOD

(*

short summary
=================
This methode replaces the Interface reference inside the collection at the given index with the given Interface.
Example:
A list of: 1 2 3 after list.replaceObjectAt(1, withObject:=4) will become: 1 4 3 and return SingleExecutionResult.SUCCESS
Example 2:
A list of: 1 2 3 after list.replaceObjectAt(3, withObject:=4) will remain: 1 2 3 and return SingleExecutionResult.ERROR

.. <legal notes>

legal notes
=================
| SPDX-FileCopyrightText: © 2022 ekvip automation GmbH <info@ekvip.de>
| SPDX-License-Identifier: Apache-2.0
| For details check: Apache-2.0_

.. _Apache-2.0: https://www.apache.org/licenses/LICENSE-2.0

.. </legal notes>

parameters
=================
:return: ``SingleExecutionResult.SUCCESS``: index valid, element at index replaced with ``withObject``
    ``SingleExecutionResult.ERROR``: ìndex out of bounds, nothing changed

*)
METHOD replaceStringContainerAt : CNM_ReturnTypes.SingleExecutionResult
VAR_INPUT
	(*the index to replace the object at*)
	index	: __XWORD;
	(*the object to be at this index instead*)
	withStringContainer	: IStringContainer;
END_VAR
replaceStringContainerAt := THIS^.list.replaceObjectAt(index := index, withObject := withStringContainer);
END_METHOD

(*

short summary
=================
This methode can replace the default sorter for a custom one. Check :ref:`IListSorter`
Can be used for performant sorting algorithms if more about the data structure is known.

.. attention:: 
	For implementations: **IListSorter is an empty interface and you should extend it with custom interfaces for each type of list.**
	For LinkedList see :ref:`ILinkedListSorter`. 
	Your implementation should then use this extended interface and the setter should check for compability. 
	
.. <legal notes>

legal notes
=================
| SPDX-FileCopyrightText: © 2022 ekvip automation GmbH <info@ekvip.de>
| SPDX-License-Identifier: Apache-2.0
| For details check: Apache-2.0_

.. _Apache-2.0: https://www.apache.org/licenses/LICENSE-2.0

.. </legal notes>

parameters
=================
:return: ``THIS^`` :ref:`IList`

*)
METHOD setSorter : CNM_CollectionInterfaces.ISortable
VAR_INPUT
	(*The instance of the sorter to be used to sort the list*)
	sorter	: CNM_CollectionInterfaces.IArrayListSorter;
END_VAR
setSorter := THIS^.list.setSorter(sorter := sorter);
END_METHOD

(*

short summary
=================
This property returns the number of elements inside this collection.

.. <legal notes>

legal notes
=================
| SPDX-FileCopyrightText: © 2022 ekvip automation GmbH <info@ekvip.de>
| SPDX-License-Identifier: Apache-2.0
| For details check: Apache-2.0_

.. _Apache-2.0: https://www.apache.org/licenses/LICENSE-2.0

.. </legal notes>

*)
PROPERTY size : __XWORD
GET
size := THIS^.list.size;
END_GET
END_PROPERTY

(*

short summary
=================
This method sorts the data structure. 
This can take many cycles and should be called until the CNM_ReturnTypes.ExecutionState is no longer ``BUSY``.

.. <legal notes>

legal notes
=================
| SPDX-FileCopyrightText: © 2022 ekvip automation GmbH <info@ekvip.de>
| SPDX-License-Identifier: Apache-2.0
| For details check: Apache-2.0_

.. _Apache-2.0: https://www.apache.org/licenses/LICENSE-2.0

.. </legal notes>

parameters
=================
:return: ``ABORTED``: While sort was pending,execute had a falling edge,
	``BUSY``: Sort is in progress
	``ERROR``: Sort was not able to finish (p.e. List changed) call sort(false) to reset
	``IDLE``: Currently no sort in progress
	``SUCCESS``: Sorting was finished 

*)
METHOD sort : CNM_ReturnTypes.SingleExecutionState
VAR_INPUT
	(*control bit to start or abort the sorting, needs to be active until the ExecutionState is SUCCESS*)
	execute	: BOOL;
END_VAR
sort := THIS^.list.sort(execute := execute);
END_METHOD

(*

short summary
=================
This method sorts the data structure. 
It uses the passed Comperator to sort the structure.
This can take many cycles and should be called until the CNM_ReturnTypes.ExecutionState is no longer ``BUSY``.

.. <legal notes>

legal notes
=================
| SPDX-FileCopyrightText: © 2022 ekvip automation GmbH <info@ekvip.de>
| SPDX-License-Identifier: Apache-2.0
| For details check: Apache-2.0_

.. _Apache-2.0: https://www.apache.org/licenses/LICENSE-2.0

.. </legal notes>

parameters
=================
:return: ``ABORTED``: While sort was pending,execute had a falling edge,
	``BUSY``: Sort is in progress
	``ERROR``: Sort was not able to finish (p.e. List changed) call sort(false) to reset
	``IDLE``: Currently no sort in progress
	``SUCCESS``: Sorting was finished 

*)
METHOD sortWithComparator : CNM_ReturnTypes.SingleExecutionState
VAR_INPUT
	(*control bit to start or abort the sorting, needs to be active until the ExecutionState is SUCCESS*)
	execute	: BOOL;
	(*the comparator that should be used for the sort. Must not be changed while sort is in process*)
	comparator	: CNM_AbstractObject.IComparator;
END_VAR
sortWithComparator := THIS^.list.sortWithComparator(execute := execute, comparator := comparator);
END_METHOD

END_FUNCTION_BLOCK

// ---- Value/Value.TcPOU
FUNCTION_BLOCK Value EXTENDS Object IMPLEMENTS IHaveValue
VAR
	myValue :LREAL;
END_VAR

(*

short summary
=================
This abstract property returns the class name of the concrete object, 
which is useful for logging/debugging purpose or to check the class name
for ``__DELETE`` in factories (sometimes it's necessary to do more 
than just to free the memory).

.. <legal notes>

legal notes
=================
| SPDX-FileCopyrightText: © 2022 ekvip automation GmbH <info@ekvip.de>
| SPDX-License-Identifier: Apache-2.0
| For details check: Apache-2.0_

.. _Apache-2.0: https://www.apache.org/licenses/LICENSE-2.0

.. </legal notes>

*)
PROPERTY className : CNM_AbstractObject.ClassName
GET
END_GET
END_PROPERTY

(*

short summary
=================
This method compares a foreign object with the own one, this is needed for sort orders.
The abstract class evaluates every object that is NULL as greater, and all other objects as equal. 

.. attention:: 
	For derivations: **If a derived class needs sorting this method must be overwritten.** 

.. <legal notes>

legal notes
=================
| SPDX-FileCopyrightText: © 2022 ekvip automation GmbH <info@ekvip.de>
| SPDX-License-Identifier: Apache-2.0
| For details check: Apache-2.0_

.. _Apache-2.0: https://www.apache.org/licenses/LICENSE-2.0

.. </legal notes>

parameters
=================
:return:``SMALLER``: ``THIS`` precedes in order,
``EQUAL``: ``THIS`` and ``object`` at the same position in order,
``GREATER``: ``THIS`` is after in order.
Checkout the library CNM_ReturnTypes.

*)
METHOD compareTo : CNM_AbstractObject.CNM_ReturnTypes.ComparationResult
VAR_INPUT
	(* foreign objet to compare*)
	object	: CNM_AbstractObject.IObject;
END_VAR
VAR
	other :IHaveValue;
END_VAR
compareTo := CNM_ReturnTypes.ComparationResult.EQUAL;

RETURN (object = 0);

IF(__QUERYINTERFACE(object, other))THEN
	IF(THIS^.value > other.value)THEN
		compareTo := CNM_ReturnTypes.ComparationResult.GREATER;
	ELSIF(THIS^.value < other.value)THEN
		compareTo := CNM_ReturnTypes.ComparationResult.SMALLER;
	END_IF
END_IF
END_METHOD

{warning 'Add property implementation'}
PROPERTY value : LREAL
GET
value := myValue;
END_GET
SET
myValue := value;
END_SET
END_PROPERTY

END_FUNCTION_BLOCK

// ---- Strings/Wrapper/LineList.TcPOU
{attribute 'enable_dynamic_creation'}
FUNCTION_BLOCK LineList EXTENDS CNM_AbstractObject.Object IMPLEMENTS ILineList
VAR
	list : CNM_Collections.ArrayList(1000);
END_VAR

(*

short summary
=================
This methode adds the given CNM_AbstractObject.IObject to the end of the list.
Example: 
Given a list that looks like this: (Head->) A B C (<- End),
calling append(D) on this list will place the D at the and,
making it the new End: (Head->) A B C D(<- End)

.. <legal notes>

legal notes
=================
| SPDX-FileCopyrightText: © 2022 ekvip automation GmbH <info@ekvip.de>
| SPDX-License-Identifier: Apache-2.0
| For details check: Apache-2.0_

.. _Apache-2.0: https://www.apache.org/licenses/LICENSE-2.0

.. </legal notes>

parameters
=================

*)
METHOD append : CNM_ReturnTypes.SingleExecutionResult
VAR_INPUT
	(*The object to be appended*)
	line	: ILine;
END_VAR
append := THIS^.list.append(object := line);
END_METHOD

(*

short summary
=================
This methode adds all elements of the given collection to the end of this list.
Example:
For the list1: A B C and list2: D E F will be after list1.appendCollection(list2):
A B C D E F. Notice the elements are still in the same order they where befor on each subsection.

.. <legal notes>

legal notes
=================
| SPDX-FileCopyrightText: © 2022 ekvip automation GmbH <info@ekvip.de>
| SPDX-License-Identifier: Apache-2.0
| For details check: Apache-2.0_

.. _Apache-2.0: https://www.apache.org/licenses/LICENSE-2.0

.. </legal notes>

parameters
=================

*)
METHOD appendCollection : CNM_ReturnTypes.SingleExecutionResult
VAR_INPUT
	(*The collection to be appended*)
	collectionToAppend	: CNM_CollectionInterfaces.ICollection;
END_VAR
appendCollection := THIS^.list.appendCollection(collectionToAppend);
END_METHOD

PROPERTY className : ClassName
GET
className := 'LineList';
END_GET
END_PROPERTY

(*

short summary
=================
This methode clears/deletes all clearable data from this object.
Example:
A list: 1 2 3 after list.clear() will have no remaining items, isEmpty = true.

.. <legal notes>

legal notes
=================
| SPDX-FileCopyrightText: © 2022 ekvip automation GmbH <info@ekvip.de>
| SPDX-License-Identifier: Apache-2.0
| For details check: Apache-2.0_

.. _Apache-2.0: https://www.apache.org/licenses/LICENSE-2.0

.. </legal notes>

parameters
=================

*)
METHOD clear
THIS^.list.clear();
END_METHOD

(*

short summary
=================
This methode checks if a given object is contained in the collection. 
The object is inside if the collection contains an object where the default comperator of the objects returns EQUAL on compareTo!

.. <legal notes>

legal notes
=================
| SPDX-FileCopyrightText: © 2022 ekvip automation GmbH <info@ekvip.de>
| SPDX-License-Identifier: Apache-2.0
| For details check: Apache-2.0_

.. _Apache-2.0: https://www.apache.org/licenses/LICENSE-2.0

.. </legal notes>

parameters
=================
:return: ``FALSE``: list does not contain an equal object
    ``TRUE``: list does contain an equal object

*)
METHOD containsEqualLine : BOOL
VAR_INPUT
	(*the object to be checked if it exists inside the collection*)
	line	: ILine;
END_VAR
containsEqualLine := THIS^.list.containsEqualObject(object := line);
END_METHOD

(*

short summary
=================
This methode checks if a given object is contained in the collection. 
The object is inside if the collection contains an object of equal hashcode!

.. <legal notes>

legal notes
=================
| SPDX-FileCopyrightText: © 2022 ekvip automation GmbH <info@ekvip.de>
| SPDX-License-Identifier: Apache-2.0
| For details check: Apache-2.0_

.. _Apache-2.0: https://www.apache.org/licenses/LICENSE-2.0

.. </legal notes>

parameters
=================
:return: ``FALSE``: list does not contain given object,
    ``TRUE``: list does contain given object

*)
METHOD containsLine : BOOL
VAR_INPUT
	(*the object to be checked if it exists inside the collection*)
	line	: ILine;
END_VAR
containsLine := THIS^.list.containsObject(object := line);
END_METHOD

{warning 'Add method implementation '}
(*

short summary
=================
This method is a self-destruction if the object was created dynamically.
If the object is a container class, the container content is destroyed with it.
The output NULL is a constant which is always NULL,
this allows a semi-pleasant notation: ``foo.deepDestruct(NULL => foo);``.

.. <legal notes>

legal notes
=================
| SPDX-FileCopyrightText: © 2022 ekvip automation GmbH <info@ekvip.de>
| SPDX-License-Identifier: Apache-2.0
| For details check: Apache-2.0_

.. _Apache-2.0: https://www.apache.org/licenses/LICENSE-2.0

.. </legal notes>

parameters
=================

InOut:
	+-----------------+------+---------+------------------------------------------+
	| Scope           | Name | Type    | Comment                                  |
	+=================+======+=========+==========================================+
	| Output CONSTANT | NULL | __XWORD | ``NULL`` is a constant which is always 0 |
	+-----------------+------+---------+------------------------------------------+

*)
METHOD deepDestruct
VAR_OUTPUT CONSTANT
	(* NULL is a constant which is always 0 *)
	NULL	: __XWORD;
END_VAR
THIS^.list.deepDestruct();
END_METHOD

(*

short summary
=================
This property returns the last object in the first and removes it from the list. Can be seen as opposite of prepend.
Example:
On a list: (Head -->) A B C, list.dequeue will return A.
Example 2:
If you call prepend(x), a dequeue right after will return x.

.. <legal notes>

legal notes
=================
| SPDX-FileCopyrightText: © 2022 ekvip automation GmbH <info@ekvip.de>
| SPDX-License-Identifier: Apache-2.0
| For details check: Apache-2.0_

.. _Apache-2.0: https://www.apache.org/licenses/LICENSE-2.0

.. </legal notes>

*)
METHOD dequeue : ILine
__QUERYINTERFACE(THIS^.list.dequeue(), dequeue);
END_METHOD

(*FB_Exit must be implemented explicitly. If there is an implementation, then the
method is called before the controller removes the code of the function block instance
(implicit call). The return value is not evaluated.*)
METHOD FB_Exit : BOOL
VAR_INPUT
	(* TRUE: the exit method is called in order to leave the instance which will be copied afterwards (online change).  *)
	bInCopyCode	: BOOL;
END_VAR
IF(THIS^.isObjectValid(THIS^.list))THEN
	THIS^.list.destruct();	
END_IF
END_METHOD

(*

short summary
=================
Method to perform a given action on all objects inside the collection.
Needs to reset the execution flag between calls.
Action to perform needs to implement :ref:`IApplier`.
Example:
You have a list of numbers: 1 2 3 and a ConcreteIncrementApplier that can take  a number and increment it. 
Calling list.forEach(TRUE, ConcreteIncrementApplier) will increment all numbers in the list, becoming: 2 3 4.

.. <legal notes>

legal notes
=================
| SPDX-FileCopyrightText: © 2022 ekvip automation GmbH <info@ekvip.de>
| SPDX-License-Identifier: Apache-2.0
| For details check: Apache-2.0_

.. _Apache-2.0: https://www.apache.org/licenses/LICENSE-2.0

.. </legal notes>

parameters
=========================
:return: CNM_ReturnTypes.ExecutionState

*)
METHOD forEach : CNM_ReturnTypes.SingleExecutionState
VAR_INPUT
	(*control bit to start or abort the forEach loop*)
	execute	: BOOL;
	(*the applier (action) to be used on all obejcts in the collection*)
	applier	: CNM_CollectionInterfaces.IApplier;
END_VAR
forEach := THIS^.list.forEach.parallel(execute := execute, applier := applier);
END_METHOD

(*

short summary
=================
This methode returns ths index of the first object that is equal to the given.
Example:
A list of: 1 2 3 after list.getIndexOf(1) will return: index=>0 and return IndexBounds.IN_BOUNDS
Example 2:
A list of: 1 2 3 after list.getIndexOf(4) will return: index=>3 and return IndexBounds.OUT_OF_BOUNDS

.. <legal notes>

legal notes
=================
| SPDX-FileCopyrightText: © 2022 ekvip automation GmbH <info@ekvip.de>
| SPDX-License-Identifier: Apache-2.0
| For details check: Apache-2.0_

.. _Apache-2.0: https://www.apache.org/licenses/LICENSE-2.0

.. </legal notes>

parameters
=================
:return: ``SingleExecutionResult.SUCCESS``: object found
    ``SingleExecutionResult.ERROR``: object couldn't be found in the list, index is undefined

*)
METHOD getIndexOf : CNM_ReturnTypes.SingleExecutionResult
VAR_INPUT
	(*the object to get the index from*)
	line	: ILine;
END_VAR
VAR_OUTPUT
	(*the index of the object inside the collection*)
	index	: __XWORD;
END_VAR
getIndexOf := THIS^.list.getIndexOf(object := line, index => index);
END_METHOD

(*

short summary
=================
This methode returns the object at the given index.
Returned objects can be modified, but not replaced! To replace an object use replaceObjectAt.
Example:
A list of: 1 2 3 after list.getObjectAt(1) will return: object=>2 and return SingleExecutionResult.SUCCESS
Example 2:
A list of: 1 2 3 after list.getObjectAt(3) will return: object=>NULL and return SingleExecutionResult.ERROR

.. <legal notes>

legal notes
=================
| SPDX-FileCopyrightText: © 2022 ekvip automation GmbH <info@ekvip.de>
| SPDX-License-Identifier: Apache-2.0
| For details check: Apache-2.0_

.. _Apache-2.0: https://www.apache.org/licenses/LICENSE-2.0

.. </legal notes>

parameters
=================
:return: ``SingleExecutionResult.SUCCESS``: index was valid
    ``SingleExecutionResult.ERROR``: index was not valid, returned object is undefined

*)
METHOD getLineAt : CNM_ReturnTypes.SingleExecutionResult
VAR_INPUT
	(*the index to access the object from*)
	index	: __XWORD;
END_VAR
VAR_OUTPUT
	(*the object at the given index*)
	line	: ILine;
END_VAR
VAR
	tmp : IObject;
END_VAR
getLineAt := THIS^.list.getObjectAt(index := index, object => tmp);
__QUERYINTERFACE(tmp, line);
END_METHOD

(*

short summary
=================
This property returns ``TRUE`` if the collection has any element.

.. <legal notes>

legal notes
=================
| SPDX-FileCopyrightText: © 2022 ekvip automation GmbH <info@ekvip.de>
| SPDX-License-Identifier: Apache-2.0
| For details check: Apache-2.0_

.. _Apache-2.0: https://www.apache.org/licenses/LICENSE-2.0

.. </legal notes>

*)
PROPERTY hasElement : BOOL
GET
hasElement := this^.list.hasElement;
END_GET
END_PROPERTY

(*

short summary
=================
This methode adds the given object at the given index. 
Will shift the other data starting at given index to the right.
List Lenght will be incremented.
Example:
A list of: 1 2 3 after list.insertObjectAt(1, object:=4) will become: 1 4 2 3 and return SingleExecutionResult.SUCCESS
Example 2:
A list of: 1 2 3 after list.insertObjectAt(3, object:=4) will become: 1 2 3 4 and return SingleExecutionResult.SUCCESS
Example 3:
A list of: 1 2 3 after list.insertObjectAt(5, object:=4) will become: 1 2 3 and return SingleExecutionResult.ERROR

.. <legal notes>

legal notes
=================
| SPDX-FileCopyrightText: © 2022 ekvip automation GmbH <info@ekvip.de>
| SPDX-License-Identifier: Apache-2.0
| For details check: Apache-2.0_

.. _Apache-2.0: https://www.apache.org/licenses/LICENSE-2.0

.. </legal notes>

parameters
=================
:return: ``SingleExecutionResult.SUCCESS``: index was valid, object inserted
    ``SingleExecutionResult.ERROR``: index out of bounds, list not changed

*)
METHOD insertLineAt : CNM_ReturnTypes.SingleExecutionResult
VAR_INPUT
	(*the index to insert the object at*)
	index	: __XWORD;
	(*the object to be added*)
	line	: ILine;
END_VAR
insertLineAt := THIS^.list.insertObjectAt(index := index, object := line);
END_METHOD

(*

short summary
=================
This method sorts the Sortable in the inverted order, so from great to low
.. <legal notes>

legal notes
=================
| SPDX-FileCopyrightText: © 2022 ekvip automation GmbH <info@ekvip.de>
| SPDX-License-Identifier: Apache-2.0
| For details check: Apache-2.0_

.. _Apache-2.0: https://www.apache.org/licenses/LICENSE-2.0

.. </legal notes>

parameters
=========================
:return: ``ABORTED``: While inverse was pending,execute had a falling edge,
	``BUSY``: Inverse is in progress
	``ERROR``: Inverse was not able to finish (p.e. List changed) call inverse(false) to reset
	``IDLE``: Currently invert is not in progress
	``SUCCESS``: Inversing was finished 
*)
METHOD inverseSort : CNM_ReturnTypes.SingleExecutionState
VAR_INPUT
	(*control bit to start or abort the inverting, needs to be active until the ExecutionState is noz longer busy*)
	execute	: BOOL;
END_VAR
inverseSort := THIS^.list.inverseSort(execute := execute);
END_METHOD

(*

short summary
=================
Inverts the order of the elements inside the object. Does not apply any kind of sorting, only reverses.

.. <legal notes>

legal notes
=================
| SPDX-FileCopyrightText: © 2022 ekvip automation GmbH <info@ekvip.de>
| SPDX-License-Identifier: Apache-2.0
| For details check: Apache-2.0_

.. _Apache-2.0: https://www.apache.org/licenses/LICENSE-2.0

.. </legal notes>

parameters
=========================

*)
METHOD invert
THIS^.list.invert();
END_METHOD

(*

short summary
=================
This property returns ``TRUE`` if the collection is empty.

.. <legal notes>

legal notes
=================
| SPDX-FileCopyrightText: © 2022 ekvip automation GmbH <info@ekvip.de>
| SPDX-License-Identifier: Apache-2.0
| For details check: Apache-2.0_

.. _Apache-2.0: https://www.apache.org/licenses/LICENSE-2.0

.. </legal notes>

*)
PROPERTY isEmpty : BOOL
GET
isEmpty := THIS^.list.isEmpty;
END_GET
END_PROPERTY

(*

